LIN {X 0,Y 446.376,Z 609.791,A -85,B 0,C 180,E1 -8740.662,E2 -8740.662} C_VEL
LIN {X 0,Y 447.077,Z 600.807,A -85,B 0,C 180,E1 -8742.253,E2 -8742.253} C_VEL
LIN {X 0,Y 447.648,Z 591.374,A -85,B 0,C 180,E1 -8743.622,E2 -8743.622} C_VEL
LIN {X 0,Y 448.423,Z 580.93,A -85,B 0,C 180,E1 -8744.872,E2 -8744.872} C_VEL
LIN {X 0,Y 449.198,Z 569.398,A -85,B 0,C 180,E1 -8746.008,E2 -8746.008} C_VEL
LIN {X 0,Y 450.087,Z 556.6,A -85,B 0,C 180,E1 -8747.025,E2 -8747.025} C_VEL
LIN {X 0,Y 450.817,Z 543.884,A -85,B 0,C 180,E1 -8747.829,E2 -8747.829} C_VEL
LIN {X 0,Y 451.423,Z 530.193,A -85,B 0,C 180,E1 -8748.495,E2 -8748.495} C_VEL
LIN {X 0,Y 451.967,Z 516.457,A -85,B 0,C 180,E1 -8748.972,E2 -8748.972} C_VEL
LIN {X 0,Y 452.276,Z 502.45,A -85,B 0,C 180,E1 -8749.282,E2 -8749.282} C_VEL
LIN {X 0,Y 453.556,Z 395.078,A -85,B 0,C 180,E1 -8750.999,E2 -8750.999} C_VEL
LIN {X 0,Y 449.146,Z 372.552,A -85,B 0,C 180,E1 -8751.608,E2 -8751.608} C_VEL
LIN {X 0,Y 449.209,Z 369.686,A -85,B 0,C 180,E1 -8752.055,E2 -8752.055} C_VEL
LIN {X 0,Y 449.824,Z 360.532,A -85,B 0,C 180,E1 -8753.724,E2 -8753.724} C_VEL
LIN {X 0,Y 448.206,Z 351.377,A -85,B 0,C 180,E1 -8755.545,E2 -8755.545} C_VEL
LIN {X 0,Y 446.531,Z 343.677,A -85,B 0,C 180,E1 -8757.158,E2 -8757.158} C_VEL
LIN {X 0,Y 446.432,Z 343.497,A -85,B 0,C 180,E1 -8760.25,E2 -8760.25} C_VEL
LIN {X 0,Y 446.449,Z 343.497,A -85,B 0,C 180,E1 -8763.454,E2 -8763.454} C_VEL
LIN {X 0,Y 446.414,Z 343.503,A -85,B 0,C 180,E1 -8766.745,E2 -8766.745} C_VEL
LIN {X 0,Y 446.46,Z 343.497,A -85,B 0,C 180,E1 -8769.526,E2 -8769.526} C_VEL
LIN {X 0,Y 446.433,Z 343.498,A -85,B 0,C 180,E1 -8772.605,E2 -8772.605} C_VEL
LIN {X 0,Y 446.456,Z 343.496,A -85,B 0,C 180,E1 -8775.104,E2 -8775.104} C_VEL
LIN {X 0,Y 446.433,Z 343.501,A -85,B 0,C 180,E1 -8778.609,E2 -8778.609} C_VEL
LIN {X 0,Y 446.448,Z 343.498,A -85,B 0,C 180,E1 -8780.973,E2 -8780.973} C_VEL
LIN {X 0,Y 446.424,Z 343.502,A -85,B 0,C 180,E1 -8784.374,E2 -8784.374} C_VEL
LIN {X 0,Y 446.427,Z 343.504,A -85,B 0,C 180,E1 -8787.639,E2 -8787.639} C_VEL
LIN {X 0,Y 446.477,Z 343.679,A -85,B 0,C 180,E1 -8790.51,E2 -8790.51} C_VEL
LIN {X 0,Y 449.215,Z 353.817,A -85,B 0,C 180,E1 -8792.262,E2 -8792.262} C_VEL
LIN {X 0,Y 450.789,Z 362.335,A -85,B 0,C 180,E1 -8793.62,E2 -8793.62} C_VEL
LIN {X 0,Y 449.985,Z 382.554,A -85,B 0,C 180,E1 -8796.53,E2 -8796.53} C_VEL
LIN {X 0,Y 449.131,Z 404.177,A -85,B 0,C 180,E1 -8799.625,E2 -8799.625} C_VEL
LIN {X 0,Y 448.594,Z 420.532,A -85,B 0,C 180,E1 -8801.952,E2 -8801.952} C_VEL
LIN {X 0,Y 450.781,Z 434.978,A -85,B 0,C 180,E1 -8802.407,E2 -8802.407} C_VEL
LIN {X 0,Y 451.257,Z 439.705,A -85,B 0,C 180,E1 -8802.531,E2 -8802.531} C_VEL
LIN {X 0,Y 449.92,Z 512.596,A -85,B 0,C 180,E1 -8803.961,E2 -8803.961} C_VEL
LIN {X 0,Y 449.624,Z 533.195,A -85,B 0,C 180,E1 -8804.387,E2 -8804.387} C_VEL
LIN {X 0,Y 449.251,Z 545.627,A -85,B 0,C 180,E1 -8804.809,E2 -8804.809} C_VEL
LIN {X 0,Y 448.731,Z 558.542,A -85,B 0,C 180,E1 -8805.43,E2 -8805.43} C_VEL
LIN {X 0,Y 448.238,Z 570.096,A -85,B 0,C 180,E1 -8806.166,E2 -8806.166} C_VEL
LIN {X 0,Y 447.634,Z 582.325,A -85,B 0,C 180,E1 -8807.169,E2 -8807.169} C_VEL
LIN {X 0,Y 447.092,Z 592.458,A -85,B 0,C 180,E1 -8808.209,E2 -8808.209} C_VEL
LIN {X 0,Y 446.575,Z 601.457,A -85,B 0,C 180,E1 -8809.344,E2 -8809.344} C_VEL
LIN {X 0,Y 446.152,Z 610.26,A -85,B 0,C 180,E1 -8810.708,E2 -8810.708} C_VEL
LIN {X 0,Y 445.834,Z 617.287,A -85,B 0,C 180,E1 -8812.072,E2 -8812.072} C_VEL
LIN {X 0,Y 445.581,Z 623.697,A -85,B 0,C 180,E1 -8813.661,E2 -8813.661} C_VEL
LIN {X 0,Y 445.499,Z 627.876,A -85,B 0,C 180,E1 -8815.023,E2 -8815.023} C_VEL
LIN {X 0,Y 445.388,Z 630.958,A -85,B 0,C 180,E1 -8816.381,E2 -8816.381} C_VEL
LIN {X 0,Y 445.405,Z 632.448,A -85,B 0,C 180,E1 -8817.287,E2 -8817.287} C_VEL
LIN {X 0,Y 445.353,Z 633.484,A -85,B 0,C 180,E1 -8818.191,E2 -8818.191} C_VEL
LIN {X 0,Y 445.316,Z 634.118,A -85,B 0,C 180,E1 -8819.096,E2 -8819.096} C_VEL
LIN {X 0,Y 445.293,Z 634.338,A -85,B 0,C 180,E1 -8820,E2 -8820} C_VEL
LIN {X 0,Y 445.316,Z 634.095,A -85,B 0,C 180,E1 -8820.904,E2 -8820.904} C_VEL
LIN {X 0,Y 445.353,Z 633.448,A -85,B 0,C 180,E1 -8821.809,E2 -8821.809} C_VEL
LIN {X 0,Y 445.405,Z 632.398,A -85,B 0,C 180,E1 -8822.713,E2 -8822.713} C_VEL
LIN {X 0,Y 445.384,Z 630.876,A -85,B 0,C 180,E1 -8823.619,E2 -8823.619} C_VEL
LIN {X 0,Y 445.493,Z 627.764,A -85,B 0,C 180,E1 -8824.978,E2 -8824.978} C_VEL
LIN {X 0,Y 445.588,Z 623.157,A -85,B 0,C 180,E1 -8826.449,E2 -8826.449} C_VEL
LIN {X 0,Y 445.797,Z 617.104,A -85,B 0,C 180,E1 -8827.929,E2 -8827.929} C_VEL
LIN {X 0,Y 446.098,Z 610.002,A -85,B 0,C 180,E1 -8829.293,E2 -8829.293} C_VEL
LIN {X 0,Y 446.496,Z 601.134,A -85,B 0,C 180,E1 -8830.658,E2 -8830.658} C_VEL
LIN {X 0,Y 446.983,Z 592.036,A -85,B 0,C 180,E1 -8831.795,E2 -8831.795} C_VEL
LIN {X 0,Y 447.491,Z 581.892,A -85,B 0,C 180,E1 -8832.823,E2 -8832.823} C_VEL
LIN {X 0,Y 447.987,Z 570.879,A -85,B 0,C 180,E1 -8833.726,E2 -8833.726} C_VEL
LIN {X 0,Y 448.466,Z 559.527,A -85,B 0,C 180,E1 -8834.463,E2 -8834.463} C_VEL
LIN {X 0,Y 448.936,Z 546.761,A -85,B 0,C 180,E1 -8835.086,E2 -8835.086} C_VEL
LIN {X 0,Y 449.3,Z 534.57,A -85,B 0,C 180,E1 -8835.509,E2 -8835.509} C_VEL
LIN {X 0,Y 449.505,Z 518.418,A -85,B 0,C 180,E1 -8835.85,E2 -8835.85} C_VEL
LIN {X 0,Y 450.479,Z 437.6,A -85,B 0,C 180,E1 -8837.331,E2 -8837.331} C_VEL
LIN {X 0,Y 448.072,Z 420.918,A -85,B 0,C 180,E1 -8837.745,E2 -8837.745} C_VEL
LIN {X 0,Y 448.866,Z 399.314,A -85,B 0,C 180,E1 -8840.867,E2 -8840.867} C_VEL
LIN {X 0,Y 449.722,Z 378.014,A -85,B 0,C 180,E1 -8843.974,E2 -8843.974} C_VEL
LIN {X 0,Y 450.347,Z 363.098,A -85,B 0,C 180,E1 -8846.159,E2 -8846.159} C_VEL
LIN {X 0,Y 449.696,Z 358.003,A -85,B 0,C 180,E1 -8846.951,E2 -8846.951} C_VEL
LIN {X 0,Y 446.503,Z 343.612,A -85,B 0,C 180,E1 -8849.316,E2 -8849.316} C_VEL
LIN {X 0,Y 446.428,Z 343.504,A -85,B 0,C 180,E1 -8852.361,E2 -8852.361} C_VEL
LIN {X 0,Y 446.425,Z 343.5,A -85,B 0,C 180,E1 -8855.626,E2 -8855.626} C_VEL
LIN {X 0,Y 446.443,Z 343.497,A -85,B 0,C 180,E1 -8859.027,E2 -8859.027} C_VEL
LIN {X 0,Y 446.439,Z 343.5,A -85,B 0,C 180,E1 -8862.277,E2 -8862.277} C_VEL
LIN {X 0,Y 446.456,Z 343.481,A -85,B 0,C 180,E1 -8865.103,E2 -8865.103} C_VEL
LIN {X 0,Y 446.434,Z 343.497,A -85,B 0,C 180,E1 -8868.609,E2 -8868.609} C_VEL
LIN {X 0,Y 446.462,Z 343.491,A -85,B 0,C 180,E1 -8870.974,E2 -8870.974} C_VEL
LIN {X 0,Y 446.426,Z 343.495,A -85,B 0,C 180,E1 -8874.374,E2 -8874.374} C_VEL
LIN {X 0,Y 446.428,Z 343.496,A -85,B 0,C 180,E1 -8877.638,E2 -8877.638} C_VEL
LIN {X 0,Y 446.454,Z 343.474,A -85,B 0,C 180,E1 -8880.79,E2 -8880.79} C_VEL
LIN {X 0,Y 446.534,Z 343.577,A -85,B 0,C 180,E1 -8882.842,E2 -8882.842} C_VEL
LIN {X 0,Y 448.194,Z 351.14,A -85,B 0,C 180,E1 -8884.454,E2 -8884.454} C_VEL
LIN {X 0,Y 449.464,Z 357.575,A -85,B 0,C 180,E1 -8885.747,E2 -8885.747} C_VEL
LIN {X 0,Y 449.036,Z 359.859,A -85,B 0,C 180,E1 -8886.151,E2 -8886.151} C_VEL
LIN {X 0,Y 446.239,Z 363.844,A -85,B 0,C 180,E1 -8886.742,E2 -8886.742} C_VEL
LIN {X 0,Y 443.163,Z 367.892,A -85,B 0,C 180,E1 -8887.336,E2 -8887.336} C_VEL
LIN {X 0,Y 442.357,Z 370.288,A -85,B 0,C 180,E1 -8887.743,E2 -8887.743} C_VEL
LIN {X 0,Y 442.345,Z 372.633,A -85,B 0,C 180,E1 -8888.092,E2 -8888.092} C_VEL
LIN {X 0,Y 446.762,Z 395.118,A -85,B 0,C 180,E1 -8888.712,E2 -8888.712} C_VEL
LIN {X 0,Y 445.847,Z 481.863,A -85,B 0,C 180,E1 -8890.129,E2 -8890.129} C_VEL
LIN {X 0,Y 445.43,Z 510.338,A -85,B 0,C 180,E1 -8890.619,E2 -8890.619} C_VEL
LIN {X 0,Y 444.898,Z 524.682,A -85,B 0,C 180,E1 -8891.044,E2 -8891.044} C_VEL
LIN {X 0,Y 444.37,Z 537.804,A -85,B 0,C 180,E1 -8891.612,E2 -8891.612} C_VEL
LIN {X 0,Y 443.61,Z 551.386,A -85,B 0,C 180,E1 -8892.393,E2 -8892.393} C_VEL
LIN {X 0,Y 442.855,Z 563.522,A -85,B 0,C 180,E1 -8893.282,E2 -8893.282} C_VEL
LIN {X 0,Y 441.938,Z 575.005,A -85,B 0,C 180,E1 -8894.314,E2 -8894.314} C_VEL
LIN {X 0,Y 441.147,Z 585.541,A -85,B 0,C 180,E1 -8895.467,E2 -8895.467} C_VEL
LIN {X 0,Y 440.361,Z 595.567,A -85,B 0,C 180,E1 -8896.791,E2 -8896.791} C_VEL
LIN {X 0,Y 439.776,Z 604.634,A -85,B 0,C 180,E1 -8898.242,E2 -8898.242} C_VEL
LIN {X 0,Y 439.211,Z 612.909,A -85,B 0,C 180,E1 -8899.861,E2 -8899.861} C_VEL
LIN {X 0,Y 438.818,Z 618.678,A -85,B 0,C 180,E1 -8901.247,E2 -8901.247} C_VEL
LIN {X 0,Y 438.526,Z 623.423,A -85,B 0,C 180,E1 -8902.633,E2 -8902.633} C_VEL
LIN {X 0,Y 438.428,Z 628.334,A -85,B 0,C 180,E1 -8904.48,E2 -8904.48} C_VEL
LIN {X 0,Y 438.275,Z 631.757,A -85,B 0,C 180,E1 -8906.321,E2 -8906.321} C_VEL
LIN {X 0,Y 438.273,Z 633.794,A -85,B 0,C 180,E1 -8908.161,E2 -8908.161} C_VEL
LIN {X 0,Y 438.205,Z 634.497,A -85,B 0,C 180,E1 -8909.999,E2 -8909.999} C_VEL
LIN {X 0,Y 438.272,Z 633.874,A -85,B 0,C 180,E1 -8911.837,E2 -8911.837} C_VEL
LIN {X 0,Y 438.274,Z 631.91,A -85,B 0,C 180,E1 -8913.676,E2 -8913.676} C_VEL
LIN {X 0,Y 438.427,Z 628.556,A -85,B 0,C 180,E1 -8915.518,E2 -8915.518} C_VEL
LIN {X 0,Y 438.521,Z 623.713,A -85,B 0,C 180,E1 -8917.365,E2 -8917.365} C_VEL
LIN {X 0,Y 438.93,Z 617.239,A -85,B 0,C 180,E1 -8919.212,E2 -8919.212} C_VEL
LIN {X 0,Y 439.321,Z 610.031,A -85,B 0,C 180,E1 -8920.833,E2 -8920.833} C_VEL
LIN {X 0,Y 440.069,Z 601.116,A -85,B 0,C 180,E1 -8922.449,E2 -8922.449} C_VEL
LIN {X 0,Y 440.7,Z 591.754,A -85,B 0,C 180,E1 -8923.839,E2 -8923.839} C_VEL
LIN {X 0,Y 441.494,Z 581.385,A -85,B 0,C 180,E1 -8925.108,E2 -8925.108} C_VEL
LIN {X 0,Y 442.384,Z 569.949,A -85,B 0,C 180,E1 -8926.259,E2 -8926.259} C_VEL
LIN {X 0,Y 443.21,Z 557.277,A -85,B 0,C 180,E1 -8927.295,E2 -8927.295} C_VEL
LIN {X 0,Y 444.099,Z 543.738,A -85,B 0,C 180,E1 -8928.165,E2 -8928.165} C_VEL
LIN {X 0,Y 444.738,Z 529.988,A -85,B 0,C 180,E1 -8928.841,E2 -8928.841} C_VEL
LIN {X 0,Y 445.286,Z 516.176,A -85,B 0,C 180,E1 -8929.325,E2 -8929.325} C_VEL
LIN {X 0,Y 445.619,Z 501.92,A -85,B 0,C 180,E1 -8929.64,E2 -8929.64} C_VEL
LIN {X 0,Y 446.91,Z 395.787,A -85,B 0,C 180,E1 -8931.364,E2 -8931.364} C_VEL
LIN {X 0,Y 442.305,Z 372.235,A -85,B 0,C 180,E1 -8932.03,E2 -8932.03} C_VEL
LIN {X 0,Y 442.902,Z 360.808,A -85,B 0,C 180,E1 -8934.116,E2 -8934.116} C_VEL
LIN {X 0,Y 440.37,Z 348.452,A -85,B 0,C 180,E1 -8936.655,E2 -8936.655} C_VEL
LIN {X 0,Y 439.506,Z 344.455,A -85,B 0,C 180,E1 -8937.555,E2 -8937.555} C_VEL
LIN {X 0,Y 439.368,Z 344.377,A -85,B 0,C 180,E1 -8940.786,E2 -8940.786} C_VEL
LIN {X 0,Y 439.384,Z 344.38,A -85,B 0,C 180,E1 -8944.042,E2 -8944.042} C_VEL
LIN {X 0,Y 439.36,Z 344.38,A -85,B 0,C 180,E1 -8947.432,E2 -8947.432} C_VEL
LIN {X 0,Y 439.423,Z 344.364,A -85,B 0,C 180,E1 -8949.852,E2 -8949.852} C_VEL
LIN {X 0,Y 439.397,Z 344.375,A -85,B 0,C 180,E1 -8952.629,E2 -8952.629} C_VEL
LIN {X 0,Y 439.397,Z 344.364,A -85,B 0,C 180,E1 -8956.032,E2 -8956.032} C_VEL
LIN {X 0,Y 439.393,Z 344.375,A -85,B 0,C 180,E1 -8959.021,E2 -8959.021} C_VEL
LIN {X 0,Y 439.385,Z 344.358,A -85,B 0,C 180,E1 -8961.604,E2 -8961.604} C_VEL
LIN {X 0,Y 439.393,Z 344.371,A -85,B 0,C 180,E1 -8964.843,E2 -8964.843} C_VEL
LIN {X 0,Y 439.366,Z 344.372,A -85,B 0,C 180,E1 -8968.139,E2 -8968.139} C_VEL
LIN {X 0,Y 439.416,Z 344.343,A -85,B 0,C 180,E1 -8971.326,E2 -8971.326} C_VEL
LIN {X 0,Y 439.403,Z 344.37,A -85,B 0,C 180,E1 -8974.415,E2 -8974.415} C_VEL
LIN {X 0,Y 439.357,Z 344.379,A -85,B 0,C 180,E1 -8977.424,E2 -8977.424} C_VEL
LIN {X 0,Y 439.431,Z 344.368,A -85,B 0,C 180,E1 -8980.662,E2 -8980.662} C_VEL
LIN {X 0,Y 439.452,Z 344.356,A -85,B 0,C 180,E1 -8984.224,E2 -8984.224} C_VEL
LIN {X 0,Y 439.498,Z 344.359,A -85,B 0,C 180,E1 -8988.002,E2 -8988.002} C_VEL
LIN {X 0,Y 439.537,Z 344.354,A -85,B 0,C 180,E1 -8991.726,E2 -8991.726} C_VEL
LIN {X 0,Y 439.614,Z 344.346,A -85,B 0,C 180,E1 -8994.496,E2 -8994.496} C_VEL
LIN {X 0,Y 439.626,Z 344.34,A -85,B 0,C 180,E1 -8998.168,E2 -8998.168} C_VEL
LIN {X 0,Y 439.755,Z 344.329,A -85,B 0,C 180,E1 -9000,E2 -9000} C_VEL
LIN {X 0,Y 439.648,Z 344.338,A -85,B 0,C 180,E1 -9002.749,E2 -9002.749} C_VEL
LIN {X 0,Y 439.61,Z 344.348,A -85,B 0,C 180,E1 -9006.425,E2 -9006.425} C_VEL
LIN {X 0,Y 439.492,Z 344.353,A -85,B 0,C 180,E1 -9009.202,E2 -9009.202} C_VEL
LIN {X 0,Y 439.493,Z 344.366,A -85,B 0,C 180,E1 -9012.727,E2 -9012.727} C_VEL
LIN {X 0,Y 439.436,Z 344.36,A -85,B 0,C 180,E1 -9016.349,E2 -9016.349} C_VEL
LIN {X 0,Y 439.393,Z 344.371,A -85,B 0,C 180,E1 -9019.627,E2 -9019.627} C_VEL
LIN {X 0,Y 439.357,Z 344.378,A -85,B 0,C 180,E1 -9022.576,E2 -9022.576} C_VEL
LIN {X 0,Y 439.403,Z 344.369,A -85,B 0,C 180,E1 -9025.585,E2 -9025.585} C_VEL
LIN {X 0,Y 439.407,Z 344.344,A -85,B 0,C 180,E1 -9028.674,E2 -9028.674} C_VEL
LIN {X 0,Y 439.361,Z 344.374,A -85,B 0,C 180,E1 -9032.031,E2 -9032.031} C_VEL
LIN {X 0,Y 439.387,Z 344.371,A -85,B 0,C 180,E1 -9035.342,E2 -9035.342} C_VEL
LIN {X 0,Y 439.389,Z 344.359,A -85,B 0,C 180,E1 -9038.594,E2 -9038.594} C_VEL
LIN {X 0,Y 439.397,Z 344.374,A -85,B 0,C 180,E1 -9041.26,E2 -9041.26} C_VEL
LIN {X 0,Y 439.403,Z 344.358,A -85,B 0,C 180,E1 -9044.729,E2 -9044.729} C_VEL
LIN {X 0,Y 439.406,Z 344.377,A -85,B 0,C 180,E1 -9047.799,E2 -9047.799} C_VEL
LIN {X 0,Y 439.446,Z 344.361,A -85,B 0,C 180,E1 -9050.231,E2 -9050.231} C_VEL
LIN {X 0,Y 439.372,Z 344.375,A -85,B 0,C 180,E1 -9053.714,E2 -9053.714} C_VEL
LIN {X 0,Y 439.371,Z 344.374,A -85,B 0,C 180,E1 -9057.056,E2 -9057.056} C_VEL
LIN {X 0,Y 439.392,Z 344.356,A -85,B 0,C 180,E1 -9060.277,E2 -9060.277} C_VEL
LIN {X 0,Y 439.514,Z 344.507,A -85,B 0,C 180,E1 -9062.516,E2 -9062.516} C_VEL
LIN {X 0,Y 442.183,Z 357.077,A -85,B 0,C 180,E1 -9065.174,E2 -9065.174} C_VEL
LIN {X 0,Y 442.975,Z 361.879,A -85,B 0,C 180,E1 -9066.137,E2 -9066.137} C_VEL
LIN {X 0,Y 442.309,Z 372.234,A -85,B 0,C 180,E1 -9068.015,E2 -9068.015} C_VEL
LIN {X 0,Y 446.811,Z 395.263,A -85,B 0,C 180,E1 -9068.667,E2 -9068.667} C_VEL
LIN {X 0,Y 445.667,Z 499.235,A -85,B 0,C 180,E1 -9070.363,E2 -9070.363} C_VEL
LIN {X 0,Y 445.33,Z 514.564,A -85,B 0,C 180,E1 -9070.677,E2 -9070.677} C_VEL
LIN {X 0,Y 444.741,Z 528.993,A -85,B 0,C 180,E1 -9071.159,E2 -9071.159} C_VEL
LIN {X 0,Y 444.135,Z 542.56,A -85,B 0,C 180,E1 -9071.811,E2 -9071.811} C_VEL
LIN {X 0,Y 443.37,Z 555.097,A -85,B 0,C 180,E1 -9072.592,E2 -9072.592} C_VEL
LIN {X 0,Y 442.576,Z 566.878,A -85,B 0,C 180,E1 -9073.511,E2 -9073.511} C_VEL
LIN {X 0,Y 441.67,Z 578.84,A -85,B 0,C 180,E1 -9074.662,E2 -9074.662} C_VEL
LIN {X 0,Y 440.831,Z 589.633,A -85,B 0,C 180,E1 -9075.93,E2 -9075.93} C_VEL
LIN {X 0,Y 440.138,Z 599.354,A -85,B 0,C 180,E1 -9077.318,E2 -9077.318} C_VEL
LIN {X 0,Y 439.576,Z 607.419,A -85,B 0,C 180,E1 -9078.707,E2 -9078.707} C_VEL
LIN {X 0,Y 439.034,Z 615.145,A -85,B 0,C 180,E1 -9080.325,E2 -9080.325} C_VEL
LIN {X 0,Y 438.709,Z 620.535,A -85,B 0,C 180,E1 -9081.712,E2 -9081.712} C_VEL
LIN {X 0,Y 438.504,Z 626.208,A -85,B 0,C 180,E1 -9083.56,E2 -9083.56} C_VEL
LIN {X 0,Y 438.33,Z 630.324,A -85,B 0,C 180,E1 -9085.403,E2 -9085.403} C_VEL
LIN {X 0,Y 438.296,Z 633.008,A -85,B 0,C 180,E1 -9087.244,E2 -9087.244} C_VEL
LIN {X 0,Y 438.228,Z 634.335,A -85,B 0,C 180,E1 -9089.082,E2 -9089.082} C_VEL
LIN {X 0,Y 438.228,Z 634.333,A -85,B 0,C 180,E1 -9090.92,E2 -9090.92} C_VEL
LIN {X 0,Y 438.296,Z 632.999,A -85,B 0,C 180,E1 -9092.758,E2 -9092.758} C_VEL
LIN {X 0,Y 438.33,Z 630.311,A -85,B 0,C 180,E1 -9094.599,E2 -9094.599} C_VEL
LIN {X 0,Y 438.465,Z 626.194,A -85,B 0,C 180,E1 -9096.443,E2 -9096.443} C_VEL
LIN {X 0,Y 438.711,Z 620.519,A -85,B 0,C 180,E1 -9098.291,E2 -9098.291} C_VEL
LIN {X 0,Y 439.118,Z 614.115,A -85,B 0,C 180,E1 -9099.908,E2 -9099.908} C_VEL
LIN {X 0,Y 439.69,Z 606.16,A -85,B 0,C 180,E1 -9101.526,E2 -9101.526} C_VEL
LIN {X 0,Y 440.286,Z 596.856,A -85,B 0,C 180,E1 -9103.068,E2 -9103.068} C_VEL
LIN {X 0,Y 440.959,Z 587.809,A -85,B 0,C 180,E1 -9104.303,E2 -9104.303} C_VEL
LIN {X 0,Y 441.827,Z 576.624,A -85,B 0,C 180,E1 -9105.572,E2 -9105.572} C_VEL
LIN {X 0,Y 442.68,Z 565.487,A -85,B 0,C 180,E1 -9106.606,E2 -9106.606} C_VEL
LIN {X 0,Y 443.502,Z 553.358,A -85,B 0,C 180,E1 -9107.524,E2 -9107.524} C_VEL
LIN {X 0,Y 444.242,Z 540.457,A -85,B 0,C 180,E1 -9108.298,E2 -9108.298} C_VEL
LIN {X 0,Y 444.831,Z 526.59,A -85,B 0,C 180,E1 -9108.929,E2 -9108.929} C_VEL
LIN {X 0,Y 445.422,Z 512.051,A -85,B 0,C 180,E1 -9109.381,E2 -9109.381} C_VEL
LIN {X 0,Y 445.768,Z 491.702,A -85,B 0,C 180,E1 -9109.755,E2 -9109.755} C_VEL
LIN {X 0,Y 446.797,Z 395.301,A -85,B 0,C 180,E1 -9111.328,E2 -9111.328} C_VEL
LIN {X 0,Y 442.295,Z 372.483,A -85,B 0,C 180,E1 -9111.964,E2 -9111.964} C_VEL
LIN {X 0,Y 442.39,Z 369.685,A -85,B 0,C 180,E1 -9112.414,E2 -9112.414} C_VEL
LIN {X 0,Y 442.925,Z 361.838,A -85,B 0,C 180,E1 -9113.868,E2 -9113.868} C_VEL
LIN {X 0,Y 441.259,Z 352.683,A -85,B 0,C 180,E1 -9115.724,E2 -9115.724} C_VEL
LIN {X 0,Y 439.48,Z 344.461,A -85,B 0,C 180,E1 -9117.501,E2 -9117.501} C_VEL
LIN {X 0,Y 439.366,Z 344.382,A -85,B 0,C 180,E1 -9120.789,E2 -9120.789} C_VEL
LIN {X 0,Y 439.392,Z 344.379,A -85,B 0,C 180,E1 -9124.044,E2 -9124.044} C_VEL
LIN {X 0,Y 439.362,Z 344.381,A -85,B 0,C 180,E1 -9126.889,E2 -9126.889} C_VEL
LIN {X 0,Y 439.406,Z 344.376,A -85,B 0,C 180,E1 -9129.85,E2 -9129.85} C_VEL
LIN {X 0,Y 439.385,Z 344.376,A -85,B 0,C 180,E1 -9132.627,E2 -9132.627} C_VEL
LIN {X 0,Y 439.404,Z 344.375,A -85,B 0,C 180,E1 -9135.271,E2 -9135.271} C_VEL
LIN {X 0,Y 439.393,Z 344.378,A -85,B 0,C 180,E1 -9138.744,E2 -9138.744} C_VEL
LIN {X 0,Y 439.379,Z 344.381,A -85,B 0,C 180,E1 -9141.608,E2 -9141.608} C_VEL
LIN {X 0,Y 439.404,Z 344.376,A -85,B 0,C 180,E1 -9144.844,E2 -9144.844} C_VEL
LIN {X 0,Y 439.378,Z 344.382,A -85,B 0,C 180,E1 -9148.14,E2 -9148.14} C_VEL
LIN {X 0,Y 439.423,Z 344.584,A -85,B 0,C 180,E1 -9150.047,E2 -9150.047} C_VEL
LIN {X 0,Y 442.588,Z 355.998,A -85,B 0,C 180,E1 -9152.067,E2 -9152.067} C_VEL
LIN {X 0,Y 444.123,Z 364.501,A -85,B 0,C 180,E1 -9153.459,E2 -9153.459} C_VEL
LIN {X 0,Y 443.117,Z 388.214,A -85,B 0,C 180,E1 -9156.913,E2 -9156.913} C_VEL
LIN {X 0,Y 442.013,Z 414.507,A -85,B 0,C 180,E1 -9160.736,E2 -9160.736} C_VEL
LIN {X 0,Y 441.811,Z 420.633,A -85,B 0,C 180,E1 -9161.599,E2 -9161.599} C_VEL
LIN {X 0,Y 444.313,Z 436.885,A -85,B 0,C 180,E1 -9162.118,E2 -9162.118} C_VEL
LIN {X 0,Y 444.594,Z 441.835,A -85,B 0,C 180,E1 -9162.242,E2 -9162.242} C_VEL
LIN {X 0,Y 443.169,Z 512.806,A -85,B 0,C 180,E1 -9163.681,E2 -9163.681} C_VEL
LIN {X 0,Y 442.841,Z 534.049,A -85,B 0,C 180,E1 -9164.141,E2 -9164.141} C_VEL
LIN {X 0,Y 442.384,Z 547.476,A -85,B 0,C 180,E1 -9164.627,E2 -9164.627} C_VEL
LIN {X 0,Y 441.875,Z 559.905,A -85,B 0,C 180,E1 -9165.257,E2 -9165.257} C_VEL
LIN {X 0,Y 441.297,Z 571.839,A -85,B 0,C 180,E1 -9166.062,E2 -9166.062} C_VEL
LIN {X 0,Y 440.724,Z 581.909,A -85,B 0,C 180,E1 -9166.91,E2 -9166.91} C_VEL
LIN {X 0,Y 440.137,Z 592.577,A -85,B 0,C 180,E1 -9168.019,E2 -9168.019} C_VEL
LIN {X 0,Y 439.586,Z 601.564,A -85,B 0,C 180,E1 -9169.172,E2 -9169.172} C_VEL
LIN {X 0,Y 439.123,Z 610.348,A -85,B 0,C 180,E1 -9170.558,E2 -9170.558} C_VEL
LIN {X 0,Y 438.777,Z 617.351,A -85,B 0,C 180,E1 -9171.943,E2 -9171.943} C_VEL
LIN {X 0,Y 438.509,Z 623.756,A -85,B 0,C 180,E1 -9173.559,E2 -9173.559} C_VEL
LIN {X 0,Y 438.434,Z 627.924,A -85,B 0,C 180,E1 -9174.942,E2 -9174.942} C_VEL
LIN {X 0,Y 438.289,Z 630.993,A -85,B 0,C 180,E1 -9176.323,E2 -9176.323} C_VEL
LIN {X 0,Y 438.317,Z 632.467,A -85,B 0,C 180,E1 -9177.243,E2 -9177.243} C_VEL
LIN {X 0,Y 438.275,Z 633.496,A -85,B 0,C 180,E1 -9178.162,E2 -9178.162} C_VEL
LIN {X 0,Y 438.232,Z 634.12,A -85,B 0,C 180,E1 -9179.081,E2 -9179.081} C_VEL
LIN {X 0,Y 438.207,Z 634.321,A -85,B 0,C 180,E1 -9180,E2 -9180} C_VEL
LIN {X 0,Y 438.231,Z 634.063,A -85,B 0,C 180,E1 -9180.919,E2 -9180.919} C_VEL
LIN {X 0,Y 438.275,Z 633.402,A -85,B 0,C 180,E1 -9181.838,E2 -9181.838} C_VEL
LIN {X 0,Y 438.302,Z 632.331,A -85,B 0,C 180,E1 -9182.757,E2 -9182.757} C_VEL
LIN {X 0,Y 438.286,Z 630.781,A -85,B 0,C 180,E1 -9183.678,E2 -9183.678} C_VEL
LIN {X 0,Y 438.406,Z 627.63,A -85,B 0,C 180,E1 -9185.058,E2 -9185.058} C_VEL
LIN {X 0,Y 438.509,Z 623.368,A -85,B 0,C 180,E1 -9186.442,E2 -9186.442} C_VEL
LIN {X 0,Y 438.74,Z 616.862,A -85,B 0,C 180,E1 -9188.057,E2 -9188.057} C_VEL
LIN {X 0,Y 439.064,Z 609.677,A -85,B 0,C 180,E1 -9189.443,E2 -9189.443} C_VEL
LIN {X 0,Y 439.461,Z 600.73,A -85,B 0,C 180,E1 -9190.831,E2 -9190.831} C_VEL
LIN {X 0,Y 440.053,Z 590.462,A -85,B 0,C 180,E1 -9192.1,E2 -9192.1} C_VEL
LIN {X 0,Y 440.627,Z 579.467,A -85,B 0,C 180,E1 -9193.193,E2 -9193.193} C_VEL
LIN {X 0,Y 441.105,Z 568.477,A -85,B 0,C 180,E1 -9194.062,E2 -9194.062} C_VEL
LIN {X 0,Y 441.661,Z 555.324,A -85,B 0,C 180,E1 -9194.868,E2 -9194.868} C_VEL
LIN {X 0,Y 442.162,Z 542.454,A -85,B 0,C 180,E1 -9195.44,E2 -9195.44} C_VEL
LIN {X 0,Y 442.502,Z 529.059,A -85,B 0,C 180,E1 -9195.842,E2 -9195.842} C_VEL
LIN {X 0,Y 443.7,Z 438.826,A -85,B 0,C 180,E1 -9197.539,E2 -9197.539} C_VEL
LIN {X 0,Y 441.144,Z 420.76,A -85,B 0,C 180,E1 -9198.009,E2 -9198.009} C_VEL
LIN {X 0,Y 441.903,Z 400.525,A -85,B 0,C 180,E1 -9200.968,E2 -9200.968} C_VEL
LIN {X 0,Y 442.899,Z 377.435,A -85,B 0,C 180,E1 -9204.367,E2 -9204.367} C_VEL
LIN {X 0,Y 443.459,Z 364.11,A -85,B 0,C 180,E1 -9206.343,E2 -9206.343} C_VEL
LIN {X 0,Y 442.324,Z 357.23,A -85,B 0,C 180,E1 -9207.437,E2 -9207.437} C_VEL
LIN {X 0,Y 439.458,Z 344.498,A -85,B 0,C 180,E1 -9209.557,E2 -9209.557} C_VEL
LIN {X 0,Y 439.378,Z 344.38,A -85,B 0,C 180,E1 -9212.946,E2 -9212.946} C_VEL
LIN {X 0,Y 439.379,Z 344.382,A -85,B 0,C 180,E1 -9216.287,E2 -9216.287} C_VEL
LIN {X 0,Y 439.407,Z 344.375,A -85,B 0,C 180,E1 -9219.849,E2 -9219.849} C_VEL
LIN {X 0,Y 439.386,Z 344.374,A -85,B 0,C 180,E1 -9222.626,E2 -9222.626} C_VEL
LIN {X 0,Y 439.405,Z 344.359,A -85,B 0,C 180,E1 -9225.27,E2 -9225.27} C_VEL
LIN {X 0,Y 439.394,Z 344.373,A -85,B 0,C 180,E1 -9228.743,E2 -9228.743} C_VEL
LIN {X 0,Y 439.39,Z 344.374,A -85,B 0,C 180,E1 -9231.605,E2 -9231.605} C_VEL
LIN {X 0,Y 439.406,Z 344.372,A -85,B 0,C 180,E1 -9234.844,E2 -9234.844} C_VEL
LIN {X 0,Y 439.378,Z 344.378,A -85,B 0,C 180,E1 -9238.139,E2 -9238.139} C_VEL
LIN {X 0,Y 439.438,Z 344.351,A -85,B 0,C 180,E1 -9241.597,E2 -9241.597} C_VEL
LIN {X 0,Y 439.486,Z 344.502,A -85,B 0,C 180,E1 -9242.563,E2 -9242.563} C_VEL
LIN {X 0,Y 442.14,Z 356.89,A -85,B 0,C 180,E1 -9245.186,E2 -9245.186} C_VEL
LIN {X 0,Y 442.91,Z 361.601,A -85,B 0,C 180,E1 -9246.131,E2 -9246.131} C_VEL
LIN {X 0,Y 442.357,Z 370.288,A -85,B 0,C 180,E1 -9247.743,E2 -9247.743} C_VEL
LIN {X 0,Y 443.121,Z 372.145,A -85,B 0,C 180,E1 -9248.027,E2 -9248.027} C_VEL
LIN {X 0,Y 446.207,Z 375.488,A -85,B 0,C 180,E1 -9248.351,E2 -9248.351} C_VEL
LIN {X 0,Y 448.816,Z 379.031,A -85,B 0,C 180,E1 -9248.543,E2 -9248.543} C_VEL
LIN {X 0,Y 449.61,Z 382.103,A -85,B 0,C 180,E1 -9248.635,E2 -9248.635} C_VEL
LIN {X 0,Y 448.993,Z 384.936,A -85,B 0,C 180,E1 -9248.645,E2 -9248.645} C_VEL
LIN {X 0,Y 446.988,Z 388.163,A -85,B 0,C 180,E1 -9248.6,E2 -9248.6} C_VEL
LIN {X 0,Y 442.3,Z 394.273,A -85,B 0,C 180,E1 -9248.472,E2 -9248.472} C_VEL
LIN {X 0,Y 441.279,Z 397.352,A -85,B 0,C 180,E1 -9248.472,E2 -9248.472} C_VEL
LIN {X 0,Y 440.234,Z 401.386,A -85,B 0,C 180,E1 -9248.488,E2 -9248.488} C_VEL
LIN {X 0,Y 438.781,Z 509.193,A -85,B 0,C 180,E1 -9250.283,E2 -9250.283} C_VEL
LIN {X 0,Y 438.219,Z 523.931,A -85,B 0,C 180,E1 -9250.713,E2 -9250.713} C_VEL
LIN {X 0,Y 437.677,Z 536.806,A -85,B 0,C 180,E1 -9251.266,E2 -9251.266} C_VEL
LIN {X 0,Y 436.895,Z 550.297,A -85,B 0,C 180,E1 -9252.038,E2 -9252.038} C_VEL
LIN {X 0,Y 436.041,Z 563.527,A -85,B 0,C 180,E1 -9253.013,E2 -9253.013} C_VEL
LIN {X 0,Y 435.082,Z 575.009,A -85,B 0,C 180,E1 -9254.06,E2 -9254.06} C_VEL
LIN {X 0,Y 434.245,Z 585.544,A -85,B 0,C 180,E1 -9255.231,E2 -9255.231} C_VEL
LIN {X 0,Y 433.372,Z 596.17,A -85,B 0,C 180,E1 -9256.662,E2 -9256.662} C_VEL
LIN {X 0,Y 432.805,Z 604.636,A -85,B 0,C 180,E1 -9258.05,E2 -9258.05} C_VEL
LIN {X 0,Y 432.156,Z 612.911,A -85,B 0,C 180,E1 -9259.694,E2 -9259.694} C_VEL
LIN {X 0,Y 431.786,Z 618.68,A -85,B 0,C 180,E1 -9261.104,E2 -9261.104} C_VEL
LIN {X 0,Y 431.479,Z 623.425,A -85,B 0,C 180,E1 -9262.512,E2 -9262.512} C_VEL
LIN {X 0,Y 431.327,Z 628.335,A -85,B 0,C 180,E1 -9264.388,E2 -9264.388} C_VEL
LIN {X 0,Y 431.182,Z 631.757,A -85,B 0,C 180,E1 -9266.261,E2 -9266.261} C_VEL
LIN {X 0,Y 431.196,Z 633.795,A -85,B 0,C 180,E1 -9268.131,E2 -9268.131} C_VEL
LIN {X 0,Y 431.121,Z 634.497,A -85,B 0,C 180,E1 -9269.999,E2 -9269.999} C_VEL
LIN {X 0,Y 431.195,Z 633.873,A -85,B 0,C 180,E1 -9271.867,E2 -9271.867} C_VEL
LIN {X 0,Y 431.181,Z 631.909,A -85,B 0,C 180,E1 -9273.737,E2 -9273.737} C_VEL
LIN {X 0,Y 431.325,Z 628.555,A -85,B 0,C 180,E1 -9275.609,E2 -9275.609} C_VEL
LIN {X 0,Y 431.474,Z 623.712,A -85,B 0,C 180,E1 -9277.486,E2 -9277.486} C_VEL
LIN {X 0,Y 431.886,Z 617.237,A -85,B 0,C 180,E1 -9279.364,E2 -9279.364} C_VEL
LIN {X 0,Y 432.317,Z 610.029,A -85,B 0,C 180,E1 -9281.011,E2 -9281.011} C_VEL
LIN {X 0,Y 432.989,Z 602.475,A -85,B 0,C 180,E1 -9282.418,E2 -9282.418} C_VEL
LIN {X 0,Y 433.637,Z 593.57,A -85,B 0,C 180,E1 -9283.806,E2 -9283.806} C_VEL
LIN {X 0,Y 434.345,Z 584.377,A -85,B 0,C 180,E1 -9285.003,E2 -9285.003} C_VEL
LIN {X 0,Y 435.204,Z 573.603,A -85,B 0,C 180,E1 -9286.173,E2 -9286.173} C_VEL
LIN {X 0,Y 436.129,Z 561.821,A -85,B 0,C 180,E1 -9287.222,E2 -9287.222} C_VEL
LIN {X 0,Y 436.972,Z 549.604,A -85,B 0,C 180,E1 -9288.101,E2 -9288.101} C_VEL
LIN {X 0,Y 437.697,Z 536.337,A -85,B 0,C 180,E1 -9288.852,E2 -9288.852} C_VEL
LIN {X 0,Y 438.339,Z 522.526,A -85,B 0,C 180,E1 -9289.431,E2 -9289.431} C_VEL
LIN {X 0,Y 438.86,Z 508.026,A -85,B 0,C 180,E1 -9289.833,E2 -9289.833} C_VEL
LIN {X 0,Y 440.267,Z 396.537,A -85,B 0,C 180,E1 -9291.689,E2 -9291.689} C_VEL
LIN {X 0,Y 435.447,Z 372.318,A -85,B 0,C 180,E1 -9292.388,E2 -9292.388} C_VEL
LIN {X 0,Y 436.06,Z 363.421,A -85,B 0,C 180,E1 -9294.012,E2 -9294.012} C_VEL
LIN {X 0,Y 434.406,Z 354.265,A -85,B 0,C 180,E1 -9295.899,E2 -9295.899} C_VEL
LIN {X 0,Y 432.444,Z 345.358,A -85,B 0,C 180,E1 -9297.854,E2 -9297.854} C_VEL
LIN {X 0,Y 432.367,Z 345.242,A -85,B 0,C 180,E1 -9300.514,E2 -9300.514} C_VEL
LIN {X 0,Y 432.356,Z 345.255,A -85,B 0,C 180,E1 -9304.002,E2 -9304.002} C_VEL
LIN {X 0,Y 432.33,Z 345.255,A -85,B 0,C 180,E1 -9307.198,E2 -9307.198} C_VEL
LIN {X 0,Y 432.353,Z 345.244,A -85,B 0,C 180,E1 -9310.182,E2 -9310.182} C_VEL
LIN {X 0,Y 432.359,Z 345.251,A -85,B 0,C 180,E1 -9313.054,E2 -9313.054} C_VEL
LIN {X 0,Y 432.371,Z 345.235,A -85,B 0,C 180,E1 -9315.657,E2 -9315.657} C_VEL
LIN {X 0,Y 432.366,Z 345.251,A -85,B 0,C 180,E1 -9318.391,E2 -9318.391} C_VEL
LIN {X 0,Y 432.345,Z 345.231,A -85,B 0,C 180,E1 -9321.851,E2 -9321.851} C_VEL
LIN {X 0,Y 432.333,Z 345.253,A -85,B 0,C 180,E1 -9325.322,E2 -9325.322} C_VEL
LIN {X 0,Y 432.315,Z 345.248,A -85,B 0,C 180,E1 -9328.653,E2 -9328.653} C_VEL
LIN {X 0,Y 432.372,Z 345.219,A -85,B 0,C 180,E1 -9331.368,E2 -9331.368} C_VEL
LIN {X 0,Y 432.359,Z 345.25,A -85,B 0,C 180,E1 -9333.967,E2 -9333.967} C_VEL
LIN {X 0,Y 432.311,Z 345.259,A -85,B 0,C 180,E1 -9337.035,E2 -9337.035} C_VEL
LIN {X 0,Y 432.377,Z 345.246,A -85,B 0,C 180,E1 -9340.514,E2 -9340.514} C_VEL
LIN {X 0,Y 432.42,Z 345.233,A -85,B 0,C 180,E1 -9343.961,E2 -9343.961} C_VEL
LIN {X 0,Y 432.471,Z 345.236,A -85,B 0,C 180,E1 -9347.804,E2 -9347.804} C_VEL
LIN {X 0,Y 432.481,Z 345.234,A -85,B 0,C 180,E1 -9351.59,E2 -9351.59} C_VEL
LIN {X 0,Y 432.59,Z 345.221,A -85,B 0,C 180,E1 -9354.406,E2 -9354.406} C_VEL
LIN {X 0,Y 432.596,Z 345.216,A -85,B 0,C 180,E1 -9358.138,E2 -9358.138} C_VEL
LIN {X 0,Y 432.726,Z 345.205,A -85,B 0,C 180,E1 -9360,E2 -9360} C_VEL
LIN {X 0,Y 432.597,Z 345.215,A -85,B 0,C 180,E1 -9362.794,E2 -9362.794} C_VEL
LIN {X 0,Y 432.564,Z 345.227,A -85,B 0,C 180,E1 -9366.53,E2 -9366.53} C_VEL
LIN {X 0,Y 432.435,Z 345.23,A -85,B 0,C 180,E1 -9369.353,E2 -9369.353} C_VEL
LIN {X 0,Y 432.434,Z 345.244,A -85,B 0,C 180,E1 -9372.812,E2 -9372.812} C_VEL
LIN {X 0,Y 432.401,Z 345.237,A -85,B 0,C 180,E1 -9376.479,E2 -9376.479} C_VEL
LIN {X 0,Y 432.331,Z 345.251,A -85,B 0,C 180,E1 -9379.961,E2 -9379.961} C_VEL
LIN {X 0,Y 432.311,Z 345.259,A -85,B 0,C 180,E1 -9382.965,E2 -9382.965} C_VEL
LIN {X 0,Y 432.358,Z 345.249,A -85,B 0,C 180,E1 -9386.033,E2 -9386.033} C_VEL
LIN {X 0,Y 432.333,Z 345.223,A -85,B 0,C 180,E1 -9389.188,E2 -9389.188} C_VEL
LIN {X 0,Y 432.314,Z 345.257,A -85,B 0,C 180,E1 -9392.444,E2 -9392.444} C_VEL
LIN {X 0,Y 432.337,Z 345.25,A -85,B 0,C 180,E1 -9395.633,E2 -9395.633} C_VEL
LIN {X 0,Y 432.351,Z 345.236,A -85,B 0,C 180,E1 -9398.719,E2 -9398.719} C_VEL
LIN {X 0,Y 432.366,Z 345.253,A -85,B 0,C 180,E1 -9401.793,E2 -9401.793} C_VEL
LIN {X 0,Y 432.371,Z 345.235,A -85,B 0,C 180,E1 -9404.343,E2 -9404.343} C_VEL
LIN {X 0,Y 432.359,Z 345.251,A -85,B 0,C 180,E1 -9407.01,E2 -9407.01} C_VEL
LIN {X 0,Y 432.352,Z 345.244,A -85,B 0,C 180,E1 -9409.818,E2 -9409.818} C_VEL
LIN {X 0,Y 432.312,Z 345.256,A -85,B 0,C 180,E1 -9413.024,E2 -9413.024} C_VEL
LIN {X 0,Y 432.355,Z 345.256,A -85,B 0,C 180,E1 -9415.998,E2 -9415.998} C_VEL
LIN {X 0,Y 432.391,Z 345.234,A -85,B 0,C 180,E1 -9419.745,E2 -9419.745} C_VEL
LIN {X 0,Y 432.459,Z 345.396,A -85,B 0,C 180,E1 -9422.213,E2 -9422.213} C_VEL
LIN {X 0,Y 435.023,Z 357.318,A -85,B 0,C 180,E1 -9424.784,E2 -9424.784} C_VEL
LIN {X 0,Y 436.077,Z 363.189,A -85,B 0,C 180,E1 -9425.989,E2 -9425.989} C_VEL
LIN {X 0,Y 435.446,Z 372.228,A -85,B 0,C 180,E1 -9427.649,E2 -9427.649} C_VEL
LIN {X 0,Y 439.189,Z 390.904,A -85,B 0,C 180,E1 -9428.203,E2 -9428.203} C_VEL
LIN {X 0,Y 440.306,Z 397.29,A -85,B 0,C 180,E1 -9428.371,E2 -9428.371} C_VEL
LIN {X 0,Y 438.809,Z 508.803,A -85,B 0,C 180,E1 -9430.226,E2 -9430.226} C_VEL
LIN {X 0,Y 438.333,Z 522.936,A -85,B 0,C 180,E1 -9430.63,E2 -9430.63} C_VEL
LIN {X 0,Y 437.787,Z 535.489,A -85,B 0,C 180,E1 -9431.152,E2 -9431.152} C_VEL
LIN {X 0,Y 437.052,Z 548.69,A -85,B 0,C 180,E1 -9431.885,E2 -9431.885} C_VEL
LIN {X 0,Y 436.225,Z 561.29,A -85,B 0,C 180,E1 -9432.782,E2 -9432.782} C_VEL
LIN {X 0,Y 435.267,Z 573.164,A -85,B 0,C 180,E1 -9433.829,E2 -9433.829} C_VEL
LIN {X 0,Y 434.365,Z 584.011,A -85,B 0,C 180,E1 -9434.998,E2 -9434.998} C_VEL
LIN {X 0,Y 433.582,Z 593.264,A -85,B 0,C 180,E1 -9436.193,E2 -9436.193} C_VEL
LIN {X 0,Y 433.036,Z 602.219,A -85,B 0,C 180,E1 -9437.583,E2 -9437.583} C_VEL
LIN {X 0,Y 432.282,Z 610.933,A -85,B 0,C 180,E1 -9439.226,E2 -9439.226} C_VEL
LIN {X 0,Y 431.886,Z 617.065,A -85,B 0,C 180,E1 -9440.636,E2 -9440.636} C_VEL
LIN {X 0,Y 431.473,Z 623.576,A -85,B 0,C 180,E1 -9442.514,E2 -9442.514} C_VEL
LIN {X 0,Y 431.407,Z 626.565,A -85,B 0,C 180,E1 -9443.588,E2 -9443.588} C_VEL
LIN {X 0,Y 431.258,Z 630.325,A -85,B 0,C 180,E1 -9445.327,E2 -9445.327} C_VEL
LIN {X 0,Y 431.193,Z 633.008,A -85,B 0,C 180,E1 -9447.199,E2 -9447.199} C_VEL
LIN {X 0,Y 431.146,Z 634.335,A -85,B 0,C 180,E1 -9449.067,E2 -9449.067} C_VEL
LIN {X 0,Y 431.146,Z 634.333,A -85,B 0,C 180,E1 -9450.935,E2 -9450.935} C_VEL
LIN {X 0,Y 431.193,Z 632.999,A -85,B 0,C 180,E1 -9452.804,E2 -9452.804} C_VEL
LIN {X 0,Y 431.259,Z 630.31,A -85,B 0,C 180,E1 -9454.675,E2 -9454.675} C_VEL
LIN {X 0,Y 431.38,Z 626.193,A -85,B 0,C 180,E1 -9456.55,E2 -9456.55} C_VEL
LIN {X 0,Y 431.653,Z 620.518,A -85,B 0,C 180,E1 -9458.427,E2 -9458.427} C_VEL
LIN {X 0,Y 432.089,Z 614.114,A -85,B 0,C 180,E1 -9460.071,E2 -9460.071} C_VEL
LIN {X 0,Y 432.689,Z 606.158,A -85,B 0,C 180,E1 -9461.715,E2 -9461.715} C_VEL
LIN {X 0,Y 433.259,Z 597.833,A -85,B 0,C 180,E1 -9463.127,E2 -9463.127} C_VEL
LIN {X 0,Y 434.043,Z 587.807,A -85,B 0,C 180,E1 -9464.536,E2 -9464.536} C_VEL
LIN {X 0,Y 434.968,Z 576.621,A -85,B 0,C 180,E1 -9465.824,E2 -9465.824} C_VEL
LIN {X 0,Y 435.974,Z 564.059,A -85,B 0,C 180,E1 -9466.99,E2 -9466.99} C_VEL
LIN {X 0,Y 436.846,Z 551.043,A -85,B 0,C 180,E1 -9467.958,E2 -9467.958} C_VEL
LIN {X 0,Y 437.658,Z 537.643,A -85,B 0,C 180,E1 -9468.734,E2 -9468.734} C_VEL
LIN {X 0,Y 438.258,Z 523.534,A -85,B 0,C 180,E1 -9469.346,E2 -9469.346} C_VEL
LIN {X 0,Y 438.758,Z 509.759,A -85,B 0,C 180,E1 -9469.749,E2 -9469.749} C_VEL
LIN {X 0,Y 440.055,Z 415.331,A -85,B 0,C 180,E1 -9471.327,E2 -9471.327} C_VEL
LIN {X 0,Y 440.204,Z 396.385,A -85,B 0,C 180,E1 -9471.645,E2 -9471.645} C_VEL
LIN {X 0,Y 435.459,Z 372.53,A -85,B 0,C 180,E1 -9472.325,E2 -9472.325} C_VEL
LIN {X 0,Y 435.594,Z 369.683,A -85,B 0,C 180,E1 -9472.783,E2 -9472.783} C_VEL
LIN {X 0,Y 436.024,Z 363.144,A -85,B 0,C 180,E1 -9474.017,E2 -9474.017} C_VEL
LIN {X 0,Y 434.102,Z 352.777,A -85,B 0,C 180,E1 -9476.161,E2 -9476.161} C_VEL
LIN {X 0,Y 432.464,Z 345.383,A -85,B 0,C 180,E1 -9477.789,E2 -9477.789} C_VEL
LIN {X 0,Y 432.326,Z 345.258,A -85,B 0,C 180,E1 -9481.347,E2 -9481.347} C_VEL
LIN {X 0,Y 432.346,Z 345.255,A -85,B 0,C 180,E1 -9484.678,E2 -9484.678} C_VEL
LIN {X 0,Y 432.35,Z 345.256,A -85,B 0,C 180,E1 -9488.15,E2 -9488.15} C_VEL
LIN {X 0,Y 432.337,Z 345.255,A -85,B 0,C 180,E1 -9491.603,E2 -9491.603} C_VEL
LIN {X 0,Y 432.338,Z 345.255,A -85,B 0,C 180,E1 -9494.348,E2 -9494.348} C_VEL
LIN {X 0,Y 432.325,Z 345.258,A -85,B 0,C 180,E1 -9497.016,E2 -9497.016} C_VEL
LIN {X 0,Y 432.338,Z 345.257,A -85,B 0,C 180,E1 -9499.821,E2 -9499.821} C_VEL
LIN {X 0,Y 432.311,Z 345.261,A -85,B 0,C 180,E1 -9503.022,E2 -9503.022} C_VEL
LIN {X 0,Y 432.364,Z 345.255,A -85,B 0,C 180,E1 -9505.997,E2 -9505.997} C_VEL
LIN {X 0,Y 432.371,Z 345.483,A -85,B 0,C 180,E1 -9509.532,E2 -9509.532} C_VEL
LIN {X 0,Y 435.322,Z 355.477,A -85,B 0,C 180,E1 -9511.379,E2 -9511.379} C_VEL
LIN {X 0,Y 437.376,Z 365.334,A -85,B 0,C 180,E1 -9513.061,E2 -9513.061} C_VEL
LIN {X 0,Y 437.195,Z 372.826,A -85,B 0,C 180,E1 -9514.187,E2 -9514.187} C_VEL
LIN {X 0,Y 436.124,Z 395.269,A -85,B 0,C 180,E1 -9517.498,E2 -9517.498} C_VEL
LIN {X 0,Y 435.077,Z 420.535,A -85,B 0,C 180,E1 -9521.199,E2 -9521.199} C_VEL
LIN {X 0,Y 437.376,Z 434.703,A -85,B 0,C 180,E1 -9521.69,E2 -9521.69} C_VEL
LIN {X 0,Y 438.063,Z 441.166,A -85,B 0,C 180,E1 -9521.878,E2 -9521.878} C_VEL
LIN {X 0,Y 436.527,Z 511.99,A -85,B 0,C 180,E1 -9523.365,E2 -9523.365} C_VEL
LIN {X 0,Y 436.089,Z 534.19,A -85,B 0,C 180,E1 -9523.859,E2 -9523.859} C_VEL
LIN {X 0,Y 435.627,Z 546.849,A -85,B 0,C 180,E1 -9524.322,E2 -9524.322} C_VEL
LIN {X 0,Y 435.082,Z 558.369,A -85,B 0,C 180,E1 -9524.902,E2 -9524.902} C_VEL
LIN {X 0,Y 434.472,Z 570.66,A -85,B 0,C 180,E1 -9525.719,E2 -9525.719} C_VEL
LIN {X 0,Y 433.79,Z 582.564,A -85,B 0,C 180,E1 -9526.735,E2 -9526.735} C_VEL
LIN {X 0,Y 433.191,Z 592.771,A -85,B 0,C 180,E1 -9527.824,E2 -9527.824} C_VEL
LIN {X 0,Y 432.607,Z 601.72,A -85,B 0,C 180,E1 -9528.995,E2 -9528.995} C_VEL
LIN {X 0,Y 432.112,Z 610.473,A -85,B 0,C 180,E1 -9530.404,E2 -9530.404} C_VEL
LIN {X 0,Y 431.736,Z 617.448,A -85,B 0,C 180,E1 -9531.811,E2 -9531.811} C_VEL
LIN {X 0,Y 431.443,Z 623.841,A -85,B 0,C 180,E1 -9533.453,E2 -9533.453} C_VEL
LIN {X 0,Y 431.368,Z 627.99,A -85,B 0,C 180,E1 -9534.859,E2 -9534.859} C_VEL
LIN {X 0,Y 431.196,Z 631.04,A -85,B 0,C 180,E1 -9536.262,E2 -9536.262} C_VEL
LIN {X 0,Y 431.214,Z 632.493,A -85,B 0,C 180,E1 -9537.198,E2 -9537.198} C_VEL
LIN {X 0,Y 431.199,Z 633.512,A -85,B 0,C 180,E1 -9538.132,E2 -9538.132} C_VEL
LIN {X 0,Y 431.15,Z 634.126,A -85,B 0,C 180,E1 -9539.066,E2 -9539.066} C_VEL
LIN {X 0,Y 431.123,Z 634.3,A -85,B 0,C 180,E1 -9540,E2 -9540} C_VEL
LIN {X 0,Y 431.15,Z 634.027,A -85,B 0,C 180,E1 -9540.934,E2 -9540.934} C_VEL
LIN {X 0,Y 431.199,Z 633.349,A -85,B 0,C 180,E1 -9541.868,E2 -9541.868} C_VEL
LIN {X 0,Y 431.199,Z 632.249,A -85,B 0,C 180,E1 -9542.803,E2 -9542.803} C_VEL
LIN {X 0,Y 431.224,Z 629.745,A -85,B 0,C 180,E1 -9544.206,E2 -9544.206} C_VEL
LIN {X 0,Y 431.342,Z 626.186,A -85,B 0,C 180,E1 -9545.61,E2 -9545.61} C_VEL
LIN {X 0,Y 431.473,Z 621.466,A -85,B 0,C 180,E1 -9547.017,E2 -9547.017} C_VEL
LIN {X 0,Y 431.782,Z 614.331,A -85,B 0,C 180,E1 -9548.659,E2 -9548.659} C_VEL
LIN {X 0,Y 432.166,Z 606.523,A -85,B 0,C 180,E1 -9550.068,E2 -9550.068} C_VEL
LIN {X 0,Y 432.558,Z 598.526,A -85,B 0,C 180,E1 -9551.243,E2 -9551.243} C_VEL
LIN {X 0,Y 433.118,Z 588.809,A -85,B 0,C 180,E1 -9552.416,E2 -9552.416} C_VEL
LIN {X 0,Y 433.656,Z 577.721,A -85,B 0,C 180,E1 -9553.494,E2 -9553.494} C_VEL
LIN {X 0,Y 434.217,Z 565.818,A -85,B 0,C 180,E1 -9554.41,E2 -9554.41} C_VEL
LIN {X 0,Y 434.759,Z 554.061,A -85,B 0,C 180,E1 -9555.11,E2 -9555.11} C_VEL
LIN {X 0,Y 435.239,Z 539.873,A -85,B 0,C 180,E1 -9555.722,E2 -9555.722} C_VEL
LIN {X 0,Y 435.625,Z 527.603,A -85,B 0,C 180,E1 -9556.069,E2 -9556.069} C_VEL
LIN {X 0,Y 436.771,Z 439.176,A -85,B 0,C 180,E1 -9557.778,E2 -9557.778} C_VEL
LIN {X 0,Y 434.196,Z 420.726,A -85,B 0,C 180,E1 -9558.268,E2 -9558.268} C_VEL
LIN {X 0,Y 435.012,Z 400.05,A -85,B 0,C 180,E1 -9561.316,E2 -9561.316} C_VEL
LIN {X 0,Y 436.071,Z 376.845,A -85,B 0,C 180,E1 -9564.774,E2 -9564.774} C_VEL
LIN {X 0,Y 436.546,Z 365.065,A -85,B 0,C 180,E1 -9566.536,E2 -9566.536} C_VEL
LIN {X 0,Y 434.552,Z 354.707,A -85,B 0,C 180,E1 -9568.214,E2 -9568.214} C_VEL
LIN {X 0,Y 432.379,Z 345.359,A -85,B 0,C 180,E1 -9569.82,E2 -9569.82} C_VEL
LIN {X 0,Y 432.345,Z 345.255,A -85,B 0,C 180,E1 -9573.552,E2 -9573.552} C_VEL
LIN {X 0,Y 432.343,Z 345.255,A -85,B 0,C 180,E1 -9575.817,E2 -9575.817} C_VEL
LIN {X 0,Y 432.332,Z 345.254,A -85,B 0,C 180,E1 -9579.345,E2 -9579.345} C_VEL
LIN {X 0,Y 432.338,Z 345.256,A -85,B 0,C 180,E1 -9581.797,E2 -9581.797} C_VEL
LIN {X 0,Y 432.339,Z 345.24,A -85,B 0,C 180,E1 -9584.347,E2 -9584.347} C_VEL
LIN {X 0,Y 432.325,Z 345.256,A -85,B 0,C 180,E1 -9587.015,E2 -9587.015} C_VEL
LIN {X 0,Y 432.338,Z 345.247,A -85,B 0,C 180,E1 -9589.82,E2 -9589.82} C_VEL
LIN {X 0,Y 432.321,Z 345.256,A -85,B 0,C 180,E1 -9593.022,E2 -9593.022} C_VEL
LIN {X 0,Y 432.365,Z 345.256,A -85,B 0,C 180,E1 -9595.996,E2 -9595.996} C_VEL
LIN {X 0,Y 432.353,Z 345.246,A -85,B 0,C 180,E1 -9599.489,E2 -9599.489} C_VEL
LIN {X 0,Y 432.483,Z 345.422,A -85,B 0,C 180,E1 -9602.278,E2 -9602.278} C_VEL
LIN {X 0,Y 435.377,Z 358.989,A -85,B 0,C 180,E1 -9605.183,E2 -9605.183} C_VEL
LIN {X 0,Y 436.014,Z 364.218,A -85,B 0,C 180,E1 -9606.235,E2 -9606.235} C_VEL
LIN {X 0,Y 435.466,Z 372.131,A -85,B 0,C 180,E1 -9607.69,E2 -9607.69} C_VEL
LIN {X 0,Y 436.658,Z 378.261,A -85,B 0,C 180,E1 -9607.901,E2 -9607.901} C_VEL
LIN {X 0,Y 440.196,Z 396.396,A -85,B 0,C 180,E1 -9608.4,E2 -9608.4} C_VEL
LIN {X 0,Y 440.234,Z 401.386,A -85,B 0,C 180,E1 -9608.488,E2 -9608.488} C_VEL
LIN {X 0,Y 439.521,Z 407.237,A -85,B 0,C 180,E1 -9608.552,E2 -9608.552} C_VEL
LIN {X 0,Y 433.887,Z 426.269,A -85,B 0,C 180,E1 -9608.591,E2 -9608.591} C_VEL
LIN {X 0,Y 433.244,Z 432.116,A -85,B 0,C 180,E1 -9608.659,E2 -9608.659} C_VEL
LIN {X 0,Y 432.118,Z 509.212,A -85,B 0,C 180,E1 -9609.966,E2 -9609.966} C_VEL
LIN {X 0,Y 431.516,Z 523.943,A -85,B 0,C 180,E1 -9610.402,E2 -9610.402} C_VEL
LIN {X 0,Y 430.97,Z 536.815,A -85,B 0,C 180,E1 -9610.964,E2 -9610.964} C_VEL
LIN {X 0,Y 430.139,Z 550.486,A -85,B 0,C 180,E1 -9611.758,E2 -9611.758} C_VEL
LIN {X 0,Y 429.229,Z 563.533,A -85,B 0,C 180,E1 -9612.735,E2 -9612.735} C_VEL
LIN {X 0,Y 428.222,Z 575.014,A -85,B 0,C 180,E1 -9613.798,E2 -9613.798} C_VEL
LIN {X 0,Y 427.375,Z 585.548,A -85,B 0,C 180,E1 -9614.988,E2 -9614.988} C_VEL
LIN {X 0,Y 426.41,Z 596.173,A -85,B 0,C 180,E1 -9616.44,E2 -9616.44} C_VEL
LIN {X 0,Y 425.835,Z 604.639,A -85,B 0,C 180,E1 -9617.852,E2 -9617.852} C_VEL
LIN {X 0,Y 425.109,Z 612.913,A -85,B 0,C 180,E1 -9619.521,E2 -9619.521} C_VEL
LIN {X 0,Y 424.742,Z 618.682,A -85,B 0,C 180,E1 -9620.955,E2 -9620.955} C_VEL
LIN {X 0,Y 424.403,Z 623.426,A -85,B 0,C 180,E1 -9622.386,E2 -9622.386} C_VEL
LIN {X 0,Y 424.236,Z 628.336,A -85,B 0,C 180,E1 -9624.294,E2 -9624.294} C_VEL
LIN {X 0,Y 424.093,Z 631.758,A -85,B 0,C 180,E1 -9626.198,E2 -9626.198} C_VEL
LIN {X 0,Y 424.121,Z 633.795,A -85,B 0,C 180,E1 -9628.1,E2 -9628.1} C_VEL
LIN {X 0,Y 424.041,Z 634.497,A -85,B 0,C 180,E1 -9629.999,E2 -9629.999} C_VEL
LIN {X 0,Y 424.12,Z 633.873,A -85,B 0,C 180,E1 -9631.898,E2 -9631.898} C_VEL
LIN {X 0,Y 424.092,Z 631.909,A -85,B 0,C 180,E1 -9633.8,E2 -9633.8} C_VEL
LIN {X 0,Y 424.232,Z 628.554,A -85,B 0,C 180,E1 -9635.703,E2 -9635.703} C_VEL
LIN {X 0,Y 424.397,Z 623.711,A -85,B 0,C 180,E1 -9637.612,E2 -9637.612} C_VEL
LIN {X 0,Y 424.717,Z 619.043,A -85,B 0,C 180,E1 -9639.043,E2 -9639.043} C_VEL
LIN {X 0,Y 425.151,Z 612.258,A -85,B 0,C 180,E1 -9640.716,E2 -9640.716} C_VEL
LIN {X 0,Y 425.789,Z 605.176,A -85,B 0,C 180,E1 -9642.147,E2 -9642.147} C_VEL
LIN {X 0,Y 426.441,Z 596.809,A -85,B 0,C 180,E1 -9643.557,E2 -9643.557} C_VEL
LIN {X 0,Y 427.305,Z 586.324,A -85,B 0,C 180,E1 -9645.012,E2 -9645.012} C_VEL
LIN {X 0,Y 428.261,Z 574.772,A -85,B 0,C 180,E1 -9646.32,E2 -9646.32} C_VEL
LIN {X 0,Y 429.233,Z 563.24,A -85,B 0,C 180,E1 -9647.385,E2 -9647.385} C_VEL
LIN {X 0,Y 430.145,Z 551.044,A -85,B 0,C 180,E1 -9648.297,E2 -9648.297} C_VEL
LIN {X 0,Y 430.907,Z 537.459,A -85,B 0,C 180,E1 -9649.098,E2 -9649.098} C_VEL
LIN {X 0,Y 431.619,Z 523.289,A -85,B 0,C 180,E1 -9649.715,E2 -9649.715} C_VEL
LIN {X 0,Y 432.149,Z 509.4,A -85,B 0,C 180,E1 -9650.123,E2 -9650.123} C_VEL
LIN {X 0,Y 433.698,Z 398.117,A -85,B 0,C 180,E1 -9652.006,E2 -9652.006} C_VEL
LIN {X 0,Y 428.974,Z 374.071,A -85,B 0,C 180,E1 -9652.688,E2 -9652.688} C_VEL
LIN {X 0,Y 428.612,Z 371.875,A -85,B 0,C 180,E1 -9652.817,E2 -9652.817} C_VEL
LIN {X 0,Y 429.179,Z 364.727,A -85,B 0,C 180,E1 -9654.165,E2 -9654.165} C_VEL
LIN {X 0,Y 426.825,Z 352.518,A -85,B 0,C 180,E1 -9656.746,E2 -9656.746} C_VEL
LIN {X 0,Y 425.374,Z 346.21,A -85,B 0,C 180,E1 -9658.19,E2 -9658.19} C_VEL
LIN {X 0,Y 425.298,Z 346.128,A -85,B 0,C 180,E1 -9660.813,E2 -9660.813} C_VEL
LIN {X 0,Y 425.308,Z 346.134,A -85,B 0,C 180,E1 -9664.287,E2 -9664.287} C_VEL
LIN {X 0,Y 425.284,Z 346.136,A -85,B 0,C 180,E1 -9667.692,E2 -9667.692} C_VEL
LIN {X 0,Y 425.297,Z 346.125,A -85,B 0,C 180,E1 -9670.523,E2 -9670.523} C_VEL
LIN {X 0,Y 425.326,Z 346.129,A -85,B 0,C 180,E1 -9673.36,E2 -9673.36} C_VEL
LIN {X 0,Y 425.325,Z 346.122,A -85,B 0,C 180,E1 -9676.637,E2 -9676.637} C_VEL
LIN {X 0,Y 425.304,Z 346.126,A -85,B 0,C 180,E1 -9679.875,E2 -9679.875} C_VEL
LIN {X 0,Y 425.279,Z 346.11,A -85,B 0,C 180,E1 -9682.486,E2 -9682.486} C_VEL
LIN {X 0,Y 425.299,Z 346.136,A -85,B 0,C 180,E1 -9685.816,E2 -9685.816} C_VEL
LIN {X 0,Y 425.291,Z 346.116,A -85,B 0,C 180,E1 -9689.236,E2 -9689.236} C_VEL
LIN {X 0,Y 425.341,Z 346.107,A -85,B 0,C 180,E1 -9692.442,E2 -9692.442} C_VEL
LIN {X 0,Y 425.345,Z 346.13,A -85,B 0,C 180,E1 -9695.602,E2 -9695.602} C_VEL
LIN {X 0,Y 425.286,Z 346.124,A -85,B 0,C 180,E1 -9698.681,E2 -9698.681} C_VEL
LIN {X 0,Y 425.323,Z 346.129,A -85,B 0,C 180,E1 -9701.702,E2 -9701.702} C_VEL
LIN {X 0,Y 425.338,Z 346.114,A -85,B 0,C 180,E1 -9704.67,E2 -9704.67} C_VEL
LIN {X 0,Y 425.42,Z 346.116,A -85,B 0,C 180,E1 -9707.598,E2 -9707.598} C_VEL
LIN {X 0,Y 425.432,Z 346.11,A -85,B 0,C 180,E1 -9711.45,E2 -9711.45} C_VEL
LIN {X 0,Y 425.547,Z 346.098,A -85,B 0,C 180,E1 -9714.313,E2 -9714.313} C_VEL
LIN {X 0,Y 425.566,Z 346.092,A -85,B 0,C 180,E1 -9718.107,E2 -9718.107} C_VEL
LIN {X 0,Y 425.696,Z 346.081,A -85,B 0,C 180,E1 -9720,E2 -9720} C_VEL
LIN {X 0,Y 425.549,Z 346.092,A -85,B 0,C 180,E1 -9722.84,E2 -9722.84} C_VEL
LIN {X 0,Y 425.522,Z 346.105,A -85,B 0,C 180,E1 -9726.639,E2 -9726.639} C_VEL
LIN {X 0,Y 425.394,Z 346.106,A -85,B 0,C 180,E1 -9729.509,E2 -9729.509} C_VEL
LIN {X 0,Y 425.393,Z 346.12,A -85,B 0,C 180,E1 -9732.911,E2 -9732.911} C_VEL
LIN {X 0,Y 425.35,Z 346.117,A -85,B 0,C 180,E1 -9736.605,E2 -9736.605} C_VEL
LIN {X 0,Y 425.318,Z 346.124,A -85,B 0,C 180,E1 -9739.636,E2 -9739.636} C_VEL
LIN {X 0,Y 425.298,Z 346.13,A -85,B 0,C 180,E1 -9743.366,E2 -9743.366} C_VEL
LIN {X 0,Y 425.339,Z 346.11,A -85,B 0,C 180,E1 -9746.845,E2 -9746.845} C_VEL
LIN {X 0,Y 425.281,Z 346.103,A -85,B 0,C 180,E1 -9749.72,E2 -9749.72} C_VEL
LIN {X 0,Y 425.273,Z 346.135,A -85,B 0,C 180,E1 -9753.049,E2 -9753.049} C_VEL
LIN {X 0,Y 425.276,Z 346.127,A -85,B 0,C 180,E1 -9755.93,E2 -9755.93} C_VEL
LIN {X 0,Y 425.304,Z 346.118,A -85,B 0,C 180,E1 -9759.047,E2 -9759.047} C_VEL
LIN {X 0,Y 425.324,Z 346.125,A -85,B 0,C 180,E1 -9762.647,E2 -9762.647} C_VEL
LIN {X 0,Y 425.327,Z 346.118,A -85,B 0,C 180,E1 -9766.055,E2 -9766.055} C_VEL
LIN {X 0,Y 425.303,Z 346.128,A -85,B 0,C 180,E1 -9768.627,E2 -9768.627} C_VEL
LIN {X 0,Y 425.318,Z 346.125,A -85,B 0,C 180,E1 -9771.105,E2 -9771.105} C_VEL
LIN {X 0,Y 425.295,Z 346.128,A -85,B 0,C 180,E1 -9774.666,E2 -9774.666} C_VEL
LIN {X 0,Y 425.269,Z 346.135,A -85,B 0,C 180,E1 -9778.075,E2 -9778.075} C_VEL
LIN {X 0,Y 425.371,Z 346.133,A -85,B 0,C 180,E1 -9781.776,E2 -9781.776} C_VEL
LIN {X 0,Y 425.408,Z 346.329,A -85,B 0,C 180,E1 -9781.913,E2 -9781.913} C_VEL
LIN {X 0,Y 428.041,Z 358.416,A -85,B 0,C 180,E1 -9784.561,E2 -9784.561} C_VEL
LIN {X 0,Y 429.159,Z 364.498,A -85,B 0,C 180,E1 -9785.834,E2 -9785.834} C_VEL
LIN {X 0,Y 428.595,Z 372.181,A -85,B 0,C 180,E1 -9787.268,E2 -9787.268} C_VEL
LIN {X 0,Y 430.861,Z 383.019,A -85,B 0,C 180,E1 -9787.62,E2 -9787.62} C_VEL
LIN {X 0,Y 433.651,Z 397.443,A -85,B 0,C 180,E1 -9788.024,E2 -9788.024} C_VEL
LIN {X 0,Y 432.273,Z 502.812,A -85,B 0,C 180,E1 -9789.79,E2 -9789.79} C_VEL
LIN {X 0,Y 431.839,Z 517.566,A -85,B 0,C 180,E1 -9790.141,E2 -9790.141} C_VEL
LIN {X 0,Y 431.193,Z 531.623,A -85,B 0,C 180,E1 -9790.668,E2 -9790.668} C_VEL
LIN {X 0,Y 430.489,Z 545.305,A -85,B 0,C 180,E1 -9791.383,E2 -9791.383} C_VEL
LIN {X 0,Y 429.631,Z 558.268,A -85,B 0,C 180,E1 -9792.263,E2 -9792.263} C_VEL
LIN {X 0,Y 428.638,Z 570.757,A -85,B 0,C 180,E1 -9793.327,E2 -9793.327} C_VEL
LIN {X 0,Y 427.688,Z 582.047,A -85,B 0,C 180,E1 -9794.514,E2 -9794.514} C_VEL
LIN {X 0,Y 426.834,Z 591.418,A -85,B 0,C 180,E1 -9795.702,E2 -9795.702} C_VEL
LIN {X 0,Y 426.119,Z 600.921,A -85,B 0,C 180,E1 -9797.149,E2 -9797.149} C_VEL
LIN {X 0,Y 425.357,Z 609.819,A -85,B 0,C 180,E1 -9798.807,E2 -9798.807} C_VEL
LIN {X 0,Y 424.835,Z 617.066,A -85,B 0,C 180,E1 -9800.479,E2 -9800.479} C_VEL
LIN {X 0,Y 424.497,Z 622.144,A -85,B 0,C 180,E1 -9801.911,E2 -9801.911} C_VEL
LIN {X 0,Y 424.33,Z 626.861,A -85,B 0,C 180,E1 -9803.594,E2 -9803.594} C_VEL
LIN {X 0,Y 424.187,Z 630.325,A -85,B 0,C 180,E1 -9805.249,E2 -9805.249} C_VEL
LIN {X 0,Y 424.09,Z 633.009,A -85,B 0,C 180,E1 -9807.152,E2 -9807.152} C_VEL
LIN {X 0,Y 424.067,Z 634.336,A -85,B 0,C 180,E1 -9809.052,E2 -9809.052} C_VEL
LIN {X 0,Y 424.067,Z 634.333,A -85,B 0,C 180,E1 -9810.951,E2 -9810.951} C_VEL
LIN {X 0,Y 424.091,Z 632.999,A -85,B 0,C 180,E1 -9812.851,E2 -9812.851} C_VEL
LIN {X 0,Y 424.187,Z 630.31,A -85,B 0,C 180,E1 -9814.753,E2 -9814.753} C_VEL
LIN {X 0,Y 424.3,Z 626.193,A -85,B 0,C 180,E1 -9816.659,E2 -9816.659} C_VEL
LIN {X 0,Y 424.614,Z 620.517,A -85,B 0,C 180,E1 -9818.568,E2 -9818.568} C_VEL
LIN {X 0,Y 425.036,Z 614.113,A -85,B 0,C 180,E1 -9820.24,E2 -9820.24} C_VEL
LIN {X 0,Y 425.691,Z 606.157,A -85,B 0,C 180,E1 -9821.911,E2 -9821.911} C_VEL
LIN {X 0,Y 426.396,Z 597,A -85,B 0,C 180,E1 -9823.478,E2 -9823.478} C_VEL
LIN {X 0,Y 427.149,Z 587.805,A -85,B 0,C 180,E1 -9824.776,E2 -9824.776} C_VEL
LIN {X 0,Y 428.122,Z 576.618,A -85,B 0,C 180,E1 -9826.083,E2 -9826.083} C_VEL
LIN {X 0,Y 429.045,Z 565.48,A -85,B 0,C 180,E1 -9827.15,E2 -9827.15} C_VEL
LIN {X 0,Y 429.947,Z 553.349,A -85,B 0,C 180,E1 -9828.095,E2 -9828.095} C_VEL
LIN {X 0,Y 430.73,Z 541.207,A -85,B 0,C 180,E1 -9828.852,E2 -9828.852} C_VEL
LIN {X 0,Y 431.379,Z 527.337,A -85,B 0,C 180,E1 -9829.512,E2 -9829.512} C_VEL
LIN {X 0,Y 432.013,Z 513.168,A -85,B 0,C 180,E1 -9829.977,E2 -9829.977} C_VEL
LIN {X 0,Y 432.382,Z 493.454,A -85,B 0,C 180,E1 -9830.362,E2 -9830.362} C_VEL
LIN {X 0,Y 433.684,Z 398.652,A -85,B 0,C 180,E1 -9831.947,E2 -9831.947} C_VEL
LIN {X 0,Y 429.934,Z 378.484,A -85,B 0,C 180,E1 -9832.505,E2 -9832.505} C_VEL
LIN {X 0,Y 428.633,Z 372.175,A -85,B 0,C 180,E1 -9832.728,E2 -9832.728} C_VEL
LIN {X 0,Y 429.129,Z 364.45,A -85,B 0,C 180,E1 -9834.17,E2 -9834.17} C_VEL
LIN {X 0,Y 427.124,Z 353.986,A -85,B 0,C 180,E1 -9836.377,E2 -9836.377} C_VEL
LIN {X 0,Y 425.388,Z 346.292,A -85,B 0,C 180,E1 -9838.091,E2 -9838.091} C_VEL
LIN {X 0,Y 425.292,Z 346.135,A -85,B 0,C 180,E1 -9840.817,E2 -9840.817} C_VEL
LIN {X 0,Y 425.317,Z 346.131,A -85,B 0,C 180,E1 -9844.289,E2 -9844.289} C_VEL
LIN {X 0,Y 425.29,Z 346.134,A -85,B 0,C 180,E1 -9847.694,E2 -9847.694} C_VEL
LIN {X 0,Y 425.284,Z 346.135,A -85,B 0,C 180,E1 -9850.521,E2 -9850.521} C_VEL
LIN {X 0,Y 425.262,Z 346.136,A -85,B 0,C 180,E1 -9853.351,E2 -9853.351} C_VEL
LIN {X 0,Y 425.262,Z 346.137,A -85,B 0,C 180,E1 -9856.65,E2 -9856.65} C_VEL
LIN {X 0,Y 425.291,Z 346.135,A -85,B 0,C 180,E1 -9859.873,E2 -9859.873} C_VEL
LIN {X 0,Y 425.283,Z 346.135,A -85,B 0,C 180,E1 -9862.489,E2 -9862.489} C_VEL
LIN {X 0,Y 425.312,Z 346.133,A -85,B 0,C 180,E1 -9865.818,E2 -9865.818} C_VEL
LIN {X 0,Y 425.309,Z 346.339,A -85,B 0,C 180,E1 -9868.948,E2 -9868.948} C_VEL
LIN {X 0,Y 428.366,Z 356.272,A -85,B 0,C 180,E1 -9870.871,E2 -9870.871} C_VEL
LIN {X 0,Y 430.777,Z 367.314,A -85,B 0,C 180,E1 -9872.818,E2 -9872.818} C_VEL
LIN {X 0,Y 430.748,Z 372.345,A -85,B 0,C 180,E1 -9873.602,E2 -9873.602} C_VEL
LIN {X 0,Y 429.5,Z 395.9,A -85,B 0,C 180,E1 -9877.131,E2 -9877.131} C_VEL
LIN {X 0,Y 428.354,Z 420.644,A -85,B 0,C 180,E1 -9880.797,E2 -9880.797} C_VEL
LIN {X 0,Y 430.981,Z 436.56,A -85,B 0,C 180,E1 -9881.362,E2 -9881.362} C_VEL
LIN {X 0,Y 431.474,Z 443.293,A -85,B 0,C 180,E1 -9881.554,E2 -9881.554} C_VEL
LIN {X 0,Y 429.882,Z 511.652,A -85,B 0,C 180,E1 -9883.039,E2 -9883.039} C_VEL
LIN {X 0,Y 429.392,Z 533.688,A -85,B 0,C 180,E1 -9883.539,E2 -9883.539} C_VEL
LIN {X 0,Y 428.886,Z 546.424,A -85,B 0,C 180,E1 -9884.008,E2 -9884.008} C_VEL
LIN {X 0,Y 428.273,Z 559.016,A -85,B 0,C 180,E1 -9884.656,E2 -9884.656} C_VEL
LIN {X 0,Y 427.632,Z 571.093,A -85,B 0,C 180,E1 -9885.485,E2 -9885.485} C_VEL
LIN {X 0,Y 426.874,Z 583.19,A -85,B 0,C 180,E1 -9886.544,E2 -9886.544} C_VEL
LIN {X 0,Y 426.261,Z 593.027,A -85,B 0,C 180,E1 -9887.623,E2 -9887.623} C_VEL
LIN {X 0,Y 425.638,Z 601.93,A -85,B 0,C 180,E1 -9888.813,E2 -9888.813} C_VEL
LIN {X 0,Y 425.114,Z 610.635,A -85,B 0,C 180,E1 -9890.244,E2 -9890.244} C_VEL
LIN {X 0,Y 424.706,Z 617.581,A -85,B 0,C 180,E1 -9891.675,E2 -9891.675} C_VEL
LIN {X 0,Y 424.389,Z 623.95,A -85,B 0,C 180,E1 -9893.343,E2 -9893.343} C_VEL
LIN {X 0,Y 424.303,Z 628.072,A -85,B 0,C 180,E1 -9894.773,E2 -9894.773} C_VEL
LIN {X 0,Y 424.108,Z 631.098,A -85,B 0,C 180,E1 -9896.199,E2 -9896.199} C_VEL
LIN {X 0,Y 424.112,Z 632.529,A -85,B 0,C 180,E1 -9897.151,E2 -9897.151} C_VEL
LIN {X 0,Y 424.125,Z 633.536,A -85,B 0,C 180,E1 -9898.101,E2 -9898.101} C_VEL
LIN {X 0,Y 424.071,Z 634.136,A -85,B 0,C 180,E1 -9899.05,E2 -9899.05} C_VEL
LIN {X 0,Y 424.043,Z 634.278,A -85,B 0,C 180,E1 -9900,E2 -9900} C_VEL
LIN {X 0,Y 424.071,Z 633.987,A -85,B 0,C 180,E1 -9900.95,E2 -9900.95} C_VEL
LIN {X 0,Y 424.124,Z 633.29,A -85,B 0,C 180,E1 -9901.899,E2 -9901.899} C_VEL
LIN {X 0,Y 424.096,Z 632.154,A -85,B 0,C 180,E1 -9902.85,E2 -9902.85} C_VEL
LIN {X 0,Y 424.147,Z 629.605,A -85,B 0,C 180,E1 -9904.276,E2 -9904.276} C_VEL
LIN {X 0,Y 424.249,Z 625.992,A -85,B 0,C 180,E1 -9905.704,E2 -9905.704} C_VEL
LIN {X 0,Y 424.415,Z 621.214,A -85,B 0,C 180,E1 -9907.134,E2 -9907.134} C_VEL
LIN {X 0,Y 424.677,Z 615.136,A -85,B 0,C 180,E1 -9908.566,E2 -9908.566} C_VEL
LIN {X 0,Y 425.057,Z 607.552,A -85,B 0,C 180,E1 -9909.998,E2 -9909.998} C_VEL
LIN {X 0,Y 425.443,Z 599.767,A -85,B 0,C 180,E1 -9911.192,E2 -9911.192} C_VEL
LIN {X 0,Y 426.055,Z 589.222,A -85,B 0,C 180,E1 -9912.504,E2 -9912.504} C_VEL
LIN {X 0,Y 426.624,Z 578.861,A -85,B 0,C 180,E1 -9913.546,E2 -9913.546} C_VEL
LIN {X 0,Y 427.202,Z 566.473,A -85,B 0,C 180,E1 -9914.53,E2 -9914.53} C_VEL
LIN {X 0,Y 427.818,Z 553.818,A -85,B 0,C 180,E1 -9915.3,E2 -9915.3} C_VEL
LIN {X 0,Y 428.292,Z 539.587,A -85,B 0,C 180,E1 -9915.923,E2 -9915.923} C_VEL
LIN {X 0,Y 428.713,Z 525.768,A -85,B 0,C 180,E1 -9916.304,E2 -9916.304} C_VEL
LIN {X 0,Y 429.967,Z 440.427,A -85,B 0,C 180,E1 -9917.99,E2 -9917.99} C_VEL
LIN {X 0,Y 427.263,Z 420.727,A -85,B 0,C 180,E1 -9918.519,E2 -9918.519} C_VEL
LIN {X 0,Y 428.068,Z 401.217,A -85,B 0,C 180,E1 -9921.426,E2 -9921.426} C_VEL
LIN {X 0,Y 429.069,Z 379.516,A -85,B 0,C 180,E1 -9924.688,E2 -9924.688} C_VEL
LIN {X 0,Y 429.594,Z 365.983,A -85,B 0,C 180,E1 -9926.737,E2 -9926.737} C_VEL
LIN {X 0,Y 427.461,Z 355.426,A -85,B 0,C 180,E1 -9928.477,E2 -9928.477} C_VEL
LIN {X 0,Y 425.338,Z 346.257,A -85,B 0,C 180,E1 -9930.057,E2 -9930.057} C_VEL
LIN {X 0,Y 425.288,Z 346.135,A -85,B 0,C 180,E1 -9933.048,E2 -9933.048} C_VEL
LIN {X 0,Y 425.288,Z 346.135,A -85,B 0,C 180,E1 -9935.928,E2 -9935.928} C_VEL
LIN {X 0,Y 425.286,Z 346.132,A -85,B 0,C 180,E1 -9939.04,E2 -9939.04} C_VEL
LIN {X 0,Y 425.295,Z 346.135,A -85,B 0,C 180,E1 -9941.958,E2 -9941.958} C_VEL
LIN {X 0,Y 425.29,Z 346.116,A -85,B 0,C 180,E1 -9945.283,E2 -9945.283} C_VEL
LIN {X 0,Y 425.28,Z 346.132,A -85,B 0,C 180,E1 -9948.621,E2 -9948.621} C_VEL
LIN {X 0,Y 425.318,Z 346.124,A -85,B 0,C 180,E1 -9951.102,E2 -9951.102} C_VEL
LIN {X 0,Y 425.306,Z 346.126,A -85,B 0,C 180,E1 -9954.664,E2 -9954.664} C_VEL
LIN {X 0,Y 425.27,Z 346.134,A -85,B 0,C 180,E1 -9958.072,E2 -9958.072} C_VEL
LIN {X 0,Y 425.387,Z 346.145,A -85,B 0,C 180,E1 -9961.875,E2 -9961.875} C_VEL
LIN {X 0,Y 425.612,Z 347.227,A -85,B 0,C 180,E1 -9962.193,E2 -9962.193} C_VEL
LIN {X 0,Y 428.428,Z 360.299,A -85,B 0,C 180,E1 -9965.012,E2 -9965.012} C_VEL
LIN {X 0,Y 429.149,Z 365.411,A -85,B 0,C 180,E1 -9966.065,E2 -9966.065} C_VEL
LIN {X 0,Y 428.624,Z 372.304,A -85,B 0,C 180,E1 -9967.331,E2 -9967.331} C_VEL
LIN {X 0,Y 433.574,Z 397.007,A -85,B 0,C 180,E1 -9968.063,E2 -9968.063} C_VEL
LIN {X 0,Y 433.244,Z 432.116,A -85,B 0,C 180,E1 -9968.659,E2 -9968.659} C_VEL
LIN {X 0,Y 432.596,Z 437.96,A -85,B 0,C 180,E1 -9968.728,E2 -9968.728} C_VEL
LIN {X 0,Y 426.941,Z 456.979,A -85,B 0,C 180,E1 -9968.768,E2 -9968.768} C_VEL
LIN {X 0,Y 426.251,Z 462.826,A -85,B 0,C 180,E1 -9968.836,E2 -9968.836} C_VEL
LIN {X 0,Y 425.436,Z 510.389,A -85,B 0,C 180,E1 -9969.669,E2 -9969.669} C_VEL
LIN {X 0,Y 424.802,Z 524.716,A -85,B 0,C 180,E1 -9970.11,E2 -9970.11} C_VEL
LIN {X 0,Y 424.149,Z 538.98,A -85,B 0,C 180,E1 -9970.766,E2 -9970.766} C_VEL
LIN {X 0,Y 423.234,Z 552.711,A -85,B 0,C 180,E1 -9971.608,E2 -9971.608} C_VEL
LIN {X 0,Y 422.311,Z 564.964,A -85,B 0,C 180,E1 -9972.568,E2 -9972.568} C_VEL
LIN {X 0,Y 421.309,Z 576.192,A -85,B 0,C 180,E1 -9973.649,E2 -9973.649} C_VEL
LIN {X 0,Y 420.315,Z 587.478,A -85,B 0,C 180,E1 -9974.978,E2 -9974.978} C_VEL
LIN {X 0,Y 419.373,Z 597.559,A -85,B 0,C 180,E1 -9976.43,E2 -9976.43} C_VEL
LIN {X 0,Y 418.735,Z 605.93,A -85,B 0,C 180,E1 -9977.888,E2 -9977.888} C_VEL
LIN {X 0,Y 418.034,Z 613.926,A -85,B 0,C 180,E1 -9979.587,E2 -9979.587} C_VEL
LIN {X 0,Y 417.561,Z 620.367,A -85,B 0,C 180,E1 -9981.286,E2 -9981.286} C_VEL
LIN {X 0,Y 417.233,Z 626.077,A -85,B 0,C 180,E1 -9983.227,E2 -9983.227} C_VEL
LIN {X 0,Y 417.118,Z 630.226,A -85,B 0,C 180,E1 -9985.166,E2 -9985.166} C_VEL
LIN {X 0,Y 416.99,Z 632.946,A -85,B 0,C 180,E1 -9987.101,E2 -9987.101} C_VEL
LIN {X 0,Y 416.991,Z 634.312,A -85,B 0,C 180,E1 -9989.033,E2 -9989.033} C_VEL
LIN {X 0,Y 416.991,Z 634.351,A -85,B 0,C 180,E1 -9990.964,E2 -9990.964} C_VEL
LIN {X 0,Y 416.989,Z 633.061,A -85,B 0,C 180,E1 -9992.897,E2 -9992.897} C_VEL
LIN {X 0,Y 417.117,Z 630.409,A -85,B 0,C 180,E1 -9994.831,E2 -9994.831} C_VEL
LIN {X 0,Y 417.231,Z 626.325,A -85,B 0,C 180,E1 -9996.77,E2 -9996.77} C_VEL
LIN {X 0,Y 417.548,Z 620.687,A -85,B 0,C 180,E1 -9998.712,E2 -9998.712} C_VEL
LIN {X 0,Y 417.986,Z 614.327,A -85,B 0,C 180,E1 -10000.412,E2 -10000.412} C_VEL
LIN {X 0,Y 418.692,Z 606.418,A -85,B 0,C 180,E1 -10002.11,E2 -10002.11} C_VEL
LIN {X 0,Y 419.371,Z 597.996,A -85,B 0,C 180,E1 -10003.593,E2 -10003.593} C_VEL
LIN {X 0,Y 420.231,Z 588.182,A -85,B 0,C 180,E1 -10005.023,E2 -10005.023} C_VEL
LIN {X 0,Y 421.252,Z 577.093,A -85,B 0,C 180,E1 -10006.35,E2 -10006.35} C_VEL
LIN {X 0,Y 422.346,Z 564.66,A -85,B 0,C 180,E1 -10007.553,E2 -10007.553} C_VEL
LIN {X 0,Y 423.307,Z 552.237,A -85,B 0,C 180,E1 -10008.519,E2 -10008.519} C_VEL
LIN {X 0,Y 424.154,Z 538.58,A -85,B 0,C 180,E1 -10009.352,E2 -10009.352} C_VEL
LIN {X 0,Y 424.87,Z 524.801,A -85,B 0,C 180,E1 -10009.978,E2 -10009.978} C_VEL
LIN {X 0,Y 425.471,Z 510.529,A -85,B 0,C 180,E1 -10010.421,E2 -10010.421} C_VEL
LIN {X 0,Y 426.155,Z 467.851,A -85,B 0,C 180,E1 -10011.177,E2 -10011.177} C_VEL
LIN {X 0,Y 426.98,Z 397.787,A -85,B 0,C 180,E1 -10012.377,E2 -10012.377} C_VEL
LIN {X 0,Y 421.866,Z 372.503,A -85,B 0,C 180,E1 -10013.14,E2 -10013.14} C_VEL
LIN {X 0,Y 421.988,Z 369.486,A -85,B 0,C 180,E1 -10013.652,E2 -10013.652} C_VEL
LIN {X 0,Y 422.282,Z 366.163,A -85,B 0,C 180,E1 -10014.297,E2 -10014.297} C_VEL
LIN {X 0,Y 419.989,Z 354.26,A -85,B 0,C 180,E1 -10016.858,E2 -10016.858} C_VEL
LIN {X 0,Y 418.364,Z 347.205,A -85,B 0,C 180,E1 -10018.466,E2 -10018.466} C_VEL
LIN {X 0,Y 418.22,Z 347.016,A -85,B 0,C 180,E1 -10021.394,E2 -10021.394} C_VEL
LIN {X 0,Y 418.262,Z 347.009,A -85,B 0,C 180,E1 -10024.579,E2 -10024.579} C_VEL
LIN {X 0,Y 418.234,Z 347.016,A -85,B 0,C 180,E1 -10027.834,E2 -10027.834} C_VEL
LIN {X 0,Y 418.262,Z 347.003,A -85,B 0,C 180,E1 -10030.941,E2 -10030.941} C_VEL
LIN {X 0,Y 418.277,Z 347,A -85,B 0,C 180,E1 -10033.739,E2 -10033.739} C_VEL
LIN {X 0,Y 418.276,Z 346.999,A -85,B 0,C 180,E1 -10036.457,E2 -10036.457} C_VEL
LIN {X 0,Y 418.26,Z 347.008,A -85,B 0,C 180,E1 -10039.122,E2 -10039.122} C_VEL
LIN {X 0,Y 418.23,Z 346.986,A -85,B 0,C 180,E1 -10042.164,E2 -10042.164} C_VEL
LIN {X 0,Y 418.257,Z 347.008,A -85,B 0,C 180,E1 -10045.419,E2 -10045.419} C_VEL
LIN {X 0,Y 418.208,Z 347.005,A -85,B 0,C 180,E1 -10048.603,E2 -10048.603} C_VEL
LIN {X 0,Y 418.286,Z 346.976,A -85,B 0,C 180,E1 -10051.936,E2 -10051.936} C_VEL
LIN {X 0,Y 418.28,Z 347.004,A -85,B 0,C 180,E1 -10055.162,E2 -10055.162} C_VEL
LIN {X 0,Y 418.226,Z 347.003,A -85,B 0,C 180,E1 -10058.303,E2 -10058.303} C_VEL
LIN {X 0,Y 418.274,Z 347.01,A -85,B 0,C 180,E1 -10061.383,E2 -10061.383} C_VEL
LIN {X 0,Y 418.292,Z 346.991,A -85,B 0,C 180,E1 -10064.405,E2 -10064.405} C_VEL
LIN {X 0,Y 418.36,Z 346.998,A -85,B 0,C 180,E1 -10067.386,E2 -10067.386} C_VEL
LIN {X 0,Y 418.351,Z 346.983,A -85,B 0,C 180,E1 -10070.329,E2 -10070.329} C_VEL
LIN {X 0,Y 418.484,Z 346.984,A -85,B 0,C 180,E1 -10073.249,E2 -10073.249} C_VEL
LIN {X 0,Y 418.335,Z 346.995,A -85,B 0,C 180,E1 -10075.181,E2 -10075.181} C_VEL
LIN {X 0,Y 418.535,Z 346.967,A -85,B 0,C 180,E1 -10078.075,E2 -10078.075} C_VEL
LIN {X 0,Y 418.665,Z 346.956,A -85,B 0,C 180,E1 -10080,E2 -10080} C_VEL
LIN {X 0,Y 418.503,Z 346.969,A -85,B 0,C 180,E1 -10082.888,E2 -10082.888} C_VEL
LIN {X 0,Y 418.484,Z 346.983,A -85,B 0,C 180,E1 -10086.751,E2 -10086.751} C_VEL
LIN {X 0,Y 418.35,Z 346.983,A -85,B 0,C 180,E1 -10089.671,E2 -10089.671} C_VEL
LIN {X 0,Y 418.344,Z 346.996,A -85,B 0,C 180,E1 -10093.007,E2 -10093.007} C_VEL
LIN {X 0,Y 418.302,Z 346.996,A -85,B 0,C 180,E1 -10096.736,E2 -10096.736} C_VEL
LIN {X 0,Y 418.261,Z 347.003,A -85,B 0,C 180,E1 -10099.791,E2 -10099.791} C_VEL
LIN {X 0,Y 418.228,Z 347.011,A -85,B 0,C 180,E1 -10102.737,E2 -10102.737} C_VEL
LIN {X 0,Y 418.264,Z 347.004,A -85,B 0,C 180,E1 -10105.904,E2 -10105.904} C_VEL
LIN {X 0,Y 418.255,Z 346.974,A -85,B 0,C 180,E1 -10109.163,E2 -10109.163} C_VEL
LIN {X 0,Y 418.248,Z 347.011,A -85,B 0,C 180,E1 -10112.845,E2 -10112.845} C_VEL
LIN {X 0,Y 418.24,Z 346.996,A -85,B 0,C 180,E1 -10116.24,E2 -10116.24} C_VEL
LIN {X 0,Y 418.258,Z 346.998,A -85,B 0,C 180,E1 -10119.681,E2 -10119.681} C_VEL
LIN {X 0,Y 418.277,Z 347.006,A -85,B 0,C 180,E1 -10122.331,E2 -10122.331} C_VEL
LIN {X 0,Y 418.267,Z 346.99,A -85,B 0,C 180,E1 -10125.115,E2 -10125.115} C_VEL
LIN {X 0,Y 418.286,Z 347.008,A -85,B 0,C 180,E1 -10127.775,E2 -10127.775} C_VEL
LIN {X 0,Y 418.261,Z 347.006,A -85,B 0,C 180,E1 -10131.561,E2 -10131.561} C_VEL
LIN {X 0,Y 418.255,Z 347.008,A -85,B 0,C 180,E1 -10135.16,E2 -10135.16} C_VEL
LIN {X 0,Y 418.245,Z 347.005,A -85,B 0,C 180,E1 -10137.474,E2 -10137.474} C_VEL
LIN {X 0,Y 418.273,Z 346.982,A -85,B 0,C 180,E1 -10140.895,E2 -10140.895} C_VEL
LIN {X 0,Y 418.328,Z 347.099,A -85,B 0,C 180,E1 -10141.531,E2 -10141.531} C_VEL
LIN {X 0,Y 420.48,Z 356.656,A -85,B 0,C 180,E1 -10143.711,E2 -10143.711} C_VEL
LIN {X 0,Y 422.248,Z 365.809,A -85,B 0,C 180,E1 -10145.675,E2 -10145.675} C_VEL
LIN {X 0,Y 421.794,Z 372.181,A -85,B 0,C 180,E1 -10146.88,E2 -10146.88} C_VEL
LIN {X 0,Y 424.184,Z 383.465,A -85,B 0,C 180,E1 -10147.256,E2 -10147.256} C_VEL
LIN {X 0,Y 427.11,Z 399.173,A -85,B 0,C 180,E1 -10147.7,E2 -10147.7} C_VEL
LIN {X 0,Y 425.59,Z 504.333,A -85,B 0,C 180,E1 -10149.49,E2 -10149.49} C_VEL
LIN {X 0,Y 425.152,Z 518.49,A -85,B 0,C 180,E1 -10149.847,E2 -10149.847} C_VEL
LIN {X 0,Y 424.44,Z 532.93,A -85,B 0,C 180,E1 -10150.41,E2 -10150.41} C_VEL
LIN {X 0,Y 423.697,Z 546.273,A -85,B 0,C 180,E1 -10151.134,E2 -10151.134} C_VEL
LIN {X 0,Y 422.848,Z 558.273,A -85,B 0,C 180,E1 -10151.969,E2 -10151.969} C_VEL
LIN {X 0,Y 421.821,Z 570.76,A -85,B 0,C 180,E1 -10153.049,E2 -10153.049} C_VEL
LIN {X 0,Y 420.808,Z 582.049,A -85,B 0,C 180,E1 -10154.254,E2 -10154.254} C_VEL
LIN {X 0,Y 419.915,Z 591.421,A -85,B 0,C 180,E1 -10155.462,E2 -10155.462} C_VEL
LIN {X 0,Y 419.122,Z 601.188,A -85,B 0,C 180,E1 -10156.977,E2 -10156.977} C_VEL
LIN {X 0,Y 418.38,Z 609.82,A -85,B 0,C 180,E1 -10158.618,E2 -10158.618} C_VEL
LIN {X 0,Y 417.798,Z 617.067,A -85,B 0,C 180,E1 -10160.317,E2 -10160.317} C_VEL
LIN {X 0,Y 417.338,Z 623.578,A -85,B 0,C 180,E1 -10162.259,E2 -10162.259} C_VEL
LIN {X 0,Y 417.26,Z 627.114,A -85,B 0,C 180,E1 -10163.591,E2 -10163.591} C_VEL
LIN {X 0,Y 417.118,Z 630.326,A -85,B 0,C 180,E1 -10165.169,E2 -10165.169} C_VEL
LIN {X 0,Y 416.989,Z 633.009,A -85,B 0,C 180,E1 -10167.103,E2 -10167.103} C_VEL
LIN {X 0,Y 416.99,Z 634.336,A -85,B 0,C 180,E1 -10169.036,E2 -10169.036} C_VEL
LIN {X 0,Y 416.99,Z 634.333,A -85,B 0,C 180,E1 -10170.967,E2 -10170.967} C_VEL
LIN {X 0,Y 416.989,Z 632.998,A -85,B 0,C 180,E1 -10172.899,E2 -10172.899} C_VEL
LIN {X 0,Y 417.117,Z 630.309,A -85,B 0,C 180,E1 -10174.834,E2 -10174.834} C_VEL
LIN {X 0,Y 417.231,Z 626.192,A -85,B 0,C 180,E1 -10176.773,E2 -10176.773} C_VEL
LIN {X 0,Y 417.551,Z 620.516,A -85,B 0,C 180,E1 -10178.714,E2 -10178.714} C_VEL
LIN {X 0,Y 418.002,Z 614.112,A -85,B 0,C 180,E1 -10180.414,E2 -10180.414} C_VEL
LIN {X 0,Y 418.713,Z 606.155,A -85,B 0,C 180,E1 -10182.112,E2 -10182.112} C_VEL
LIN {X 0,Y 419.416,Z 597.529,A -85,B 0,C 180,E1 -10183.619,E2 -10183.619} C_VEL
LIN {X 0,Y 420.257,Z 587.803,A -85,B 0,C 180,E1 -10185.024,E2 -10185.024} C_VEL
LIN {X 0,Y 421.262,Z 576.615,A -85,B 0,C 180,E1 -10186.353,E2 -10186.353} C_VEL
LIN {X 0,Y 422.38,Z 564.051,A -85,B 0,C 180,E1 -10187.554,E2 -10187.554} C_VEL
LIN {X 0,Y 423.313,Z 551.436,A -85,B 0,C 180,E1 -10188.524,E2 -10188.524} C_VEL
LIN {X 0,Y 424.235,Z 537.631,A -85,B 0,C 180,E1 -10189.35,E2 -10189.35} C_VEL
LIN {X 0,Y 424.875,Z 524.28,A -85,B 0,C 180,E1 -10189.949,E2 -10189.949} C_VEL
LIN {X 0,Y 425.436,Z 509.735,A -85,B 0,C 180,E1 -10190.394,E2 -10190.394} C_VEL
LIN {X 0,Y 426.818,Z 420.123,A -85,B 0,C 180,E1 -10191.937,E2 -10191.937} C_VEL
LIN {X 0,Y 426.956,Z 397.886,A -85,B 0,C 180,E1 -10192.325,E2 -10192.325} C_VEL
LIN {X 0,Y 421.88,Z 372.421,A -85,B 0,C 180,E1 -10193.093,E2 -10193.093} C_VEL
LIN {X 0,Y 422.093,Z 368.503,A -85,B 0,C 180,E1 -10193.789,E2 -10193.789} C_VEL
LIN {X 0,Y 422.23,Z 365.757,A -85,B 0,C 180,E1 -10194.329,E2 -10194.329} C_VEL
LIN {X 0,Y 419.884,Z 353.984,A -85,B 0,C 180,E1 -10196.868,E2 -10196.868} C_VEL
LIN {X 0,Y 418.331,Z 347.067,A -85,B 0,C 180,E1 -10198.471,E2 -10198.471} C_VEL
LIN {X 0,Y 418.216,Z 347.015,A -85,B 0,C 180,E1 -10201.397,E2 -10201.397} C_VEL
LIN {X 0,Y 418.271,Z 347.008,A -85,B 0,C 180,E1 -10204.581,E2 -10204.581} C_VEL
LIN {X 0,Y 418.238,Z 347.012,A -85,B 0,C 180,E1 -10207.835,E2 -10207.835} C_VEL
LIN {X 0,Y 418.226,Z 347.012,A -85,B 0,C 180,E1 -10210.949,E2 -10210.949} C_VEL
LIN {X 0,Y 418.214,Z 347.017,A -85,B 0,C 180,E1 -10213.73,E2 -10213.73} C_VEL
LIN {X 0,Y 418.213,Z 347.015,A -85,B 0,C 180,E1 -10216.449,E2 -10216.449} C_VEL
LIN {X 0,Y 418.228,Z 347.015,A -85,B 0,C 180,E1 -10219.131,E2 -10219.131} C_VEL
LIN {X 0,Y 418.233,Z 347.013,A -85,B 0,C 180,E1 -10222.167,E2 -10222.167} C_VEL
LIN {X 0,Y 418.27,Z 347.011,A -85,B 0,C 180,E1 -10225.42,E2 -10225.42} C_VEL
LIN {X 0,Y 418.261,Z 347.161,A -85,B 0,C 180,E1 -10228.29,E2 -10228.29} C_VEL
LIN {X 0,Y 421.759,Z 358.286,A -85,B 0,C 180,E1 -10230.55,E2 -10230.55} C_VEL
LIN {X 0,Y 423.97,Z 368.102,A -85,B 0,C 180,E1 -10232.345,E2 -10232.345} C_VEL
LIN {X 0,Y 424.371,Z 371.404,A -85,B 0,C 180,E1 -10232.908,E2 -10232.908} C_VEL
LIN {X 0,Y 422.903,Z 396.655,A -85,B 0,C 180,E1 -10236.753,E2 -10236.753} C_VEL
LIN {X 0,Y 421.677,Z 420.476,A -85,B 0,C 180,E1 -10240.339,E2 -10240.339} C_VEL
LIN {X 0,Y 424.25,Z 435.332,A -85,B 0,C 180,E1 -10240.915,E2 -10240.915} C_VEL
LIN {X 0,Y 425.013,Z 443.298,A -85,B 0,C 180,E1 -10241.164,E2 -10241.164} C_VEL
LIN {X 0,Y 423.152,Z 513.168,A -85,B 0,C 180,E1 -10242.73,E2 -10242.73} C_VEL
LIN {X 0,Y 422.693,Z 534.419,A -85,B 0,C 180,E1 -10243.24,E2 -10243.24} C_VEL
LIN {X 0,Y 422.14,Z 547.518,A -85,B 0,C 180,E1 -10243.746,E2 -10243.746} C_VEL
LIN {X 0,Y 421.475,Z 559.782,A -85,B 0,C 180,E1 -10244.402,E2 -10244.402} C_VEL
LIN {X 0,Y 420.798,Z 571.634,A -85,B 0,C 180,E1 -10245.244,E2 -10245.244} C_VEL
LIN {X 0,Y 420.038,Z 582.861,A -85,B 0,C 180,E1 -10246.244,E2 -10246.244} C_VEL
LIN {X 0,Y 419.351,Z 593.349,A -85,B 0,C 180,E1 -10247.416,E2 -10247.416} C_VEL
LIN {X 0,Y 418.681,Z 602.193,A -85,B 0,C 180,E1 -10248.625,E2 -10248.625} C_VEL
LIN {X 0,Y 418.127,Z 610.842,A -85,B 0,C 180,E1 -10250.079,E2 -10250.079} C_VEL
LIN {X 0,Y 417.687,Z 617.748,A -85,B 0,C 180,E1 -10251.534,E2 -10251.534} C_VEL
LIN {X 0,Y 417.319,Z 624.083,A -85,B 0,C 180,E1 -10253.23,E2 -10253.23} C_VEL
LIN {X 0,Y 417.218,Z 628.17,A -85,B 0,C 180,E1 -10254.684,E2 -10254.684} C_VEL
LIN {X 0,Y 417.024,Z 631.168,A -85,B 0,C 180,E1 -10256.135,E2 -10256.135} C_VEL
LIN {X 0,Y 417.011,Z 632.574,A -85,B 0,C 180,E1 -10257.102,E2 -10257.102} C_VEL
LIN {X 0,Y 417.034,Z 633.566,A -85,B 0,C 180,E1 -10258.069,E2 -10258.069} C_VEL
LIN {X 0,Y 416.994,Z 634.145,A -85,B 0,C 180,E1 -10259.034,E2 -10259.034} C_VEL
LIN {X 0,Y 416.965,Z 634.254,A -85,B 0,C 180,E1 -10260,E2 -10260} C_VEL
LIN {X 0,Y 416.994,Z 633.944,A -85,B 0,C 180,E1 -10260.966,E2 -10260.966} C_VEL
LIN {X 0,Y 417.033,Z 633.226,A -85,B 0,C 180,E1 -10261.932,E2 -10261.932} C_VEL
LIN {X 0,Y 416.995,Z 632.047,A -85,B 0,C 180,E1 -10262.898,E2 -10262.898} C_VEL
LIN {X 0,Y 417.075,Z 629.448,A -85,B 0,C 180,E1 -10264.349,E2 -10264.349} C_VEL
LIN {X 0,Y 417.159,Z 625.776,A -85,B 0,C 180,E1 -10265.802,E2 -10265.802} C_VEL
LIN {X 0,Y 417.352,Z 620.931,A -85,B 0,C 180,E1 -10267.256,E2 -10267.256} C_VEL
LIN {X 0,Y 417.612,Z 614.776,A -85,B 0,C 180,E1 -10268.712,E2 -10268.712} C_VEL
LIN {X 0,Y 418,Z 607.088,A -85,B 0,C 180,E1 -10270.168,E2 -10270.168} C_VEL
LIN {X 0,Y 418.546,Z 597.406,A -85,B 0,C 180,E1 -10271.625,E2 -10271.625} C_VEL
LIN {X 0,Y 419.152,Z 587.421,A -85,B 0,C 180,E1 -10272.836,E2 -10272.836} C_VEL
LIN {X 0,Y 419.767,Z 576.214,A -85,B 0,C 180,E1 -10273.926,E2 -10273.926} C_VEL
LIN {X 0,Y 420.281,Z 565.341,A -85,B 0,C 180,E1 -10274.774,E2 -10274.774} C_VEL
LIN {X 0,Y 420.849,Z 553.416,A -85,B 0,C 180,E1 -10275.497,E2 -10275.497} C_VEL
LIN {X 0,Y 421.328,Z 539.882,A -85,B 0,C 180,E1 -10276.1,E2 -10276.1} C_VEL
LIN {X 0,Y 421.772,Z 526.392,A -85,B 0,C 180,E1 -10276.487,E2 -10276.487} C_VEL
LIN {X 0,Y 423.083,Z 441.169,A -85,B 0,C 180,E1 -10278.22,E2 -10278.22} C_VEL
LIN {X 0,Y 420.334,Z 420.766,A -85,B 0,C 180,E1 -10278.776,E2 -10278.776} C_VEL
LIN {X 0,Y 421.28,Z 398.999,A -85,B 0,C 180,E1 -10282.046,E2 -10282.046} C_VEL
LIN {X 0,Y 422.263,Z 378.819,A -85,B 0,C 180,E1 -10285.114,E2 -10285.114} C_VEL
LIN {X 0,Y 422.762,Z 368.635,A -85,B 0,C 180,E1 -10286.67,E2 -10286.67} C_VEL
LIN {X 0,Y 421.983,Z 363.386,A -85,B 0,C 180,E1 -10287.527,E2 -10287.527} C_VEL
LIN {X 0,Y 418.32,Z 347.176,A -85,B 0,C 180,E1 -10290.297,E2 -10290.297} C_VEL
LIN {X 0,Y 418.254,Z 347.011,A -85,B 0,C 180,E1 -10293.677,E2 -10293.677} C_VEL
LIN {X 0,Y 418.245,Z 347.01,A -85,B 0,C 180,E1 -10297.224,E2 -10297.224} C_VEL
LIN {X 0,Y 418.25,Z 347.01,A -85,B 0,C 180,E1 -10299.682,E2 -10299.682} C_VEL
LIN {X 0,Y 418.235,Z 347.012,A -85,B 0,C 180,E1 -10302.321,E2 -10302.321} C_VEL
LIN {X 0,Y 418.241,Z 346.992,A -85,B 0,C 180,E1 -10305.108,E2 -10305.108} C_VEL
LIN {X 0,Y 418.246,Z 347.013,A -85,B 0,C 180,E1 -10307.766,E2 -10307.766} C_VEL
LIN {X 0,Y 418.264,Z 347.005,A -85,B 0,C 180,E1 -10311.558,E2 -10311.558} C_VEL
LIN {X 0,Y 418.265,Z 347.006,A -85,B 0,C 180,E1 -10315.158,E2 -10315.158} C_VEL
LIN {X 0,Y 418.251,Z 347.004,A -85,B 0,C 180,E1 -10317.471,E2 -10317.471} C_VEL
LIN {X 0,Y 418.274,Z 346.982,A -85,B 0,C 180,E1 -10320.895,E2 -10320.895} C_VEL
LIN {X 0,Y 418.358,Z 347.117,A -85,B 0,C 180,E1 -10321.599,E2 -10321.599} C_VEL
LIN {X 0,Y 421.046,Z 359.285,A -85,B 0,C 180,E1 -10324.337,E2 -10324.337} C_VEL
LIN {X 0,Y 422.189,Z 365.532,A -85,B 0,C 180,E1 -10325.668,E2 -10325.668} C_VEL
LIN {X 0,Y 421.841,Z 372.149,A -85,B 0,C 180,E1 -10326.929,E2 -10326.929} C_VEL
LIN {X 0,Y 423.213,Z 378.753,A -85,B 0,C 180,E1 -10327.168,E2 -10327.168} C_VEL
LIN {X 0,Y 427.007,Z 398.068,A -85,B 0,C 180,E1 -10327.726,E2 -10327.726} C_VEL
LIN {X 0,Y 426.251,Z 462.826,A -85,B 0,C 180,E1 -10328.836,E2 -10328.836} C_VEL
LIN {X 0,Y 425.57,Z 468.669,A -85,B 0,C 180,E1 -10328.904,E2 -10328.904} C_VEL
LIN {X 0,Y 419.885,Z 487.675,A -85,B 0,C 180,E1 -10328.945,E2 -10328.945} C_VEL
LIN {X 0,Y 419.155,Z 493.521,A -85,B 0,C 180,E1 -10329.012,E2 -10329.012} C_VEL
LIN {X 0,Y 418.691,Z 512.687,A -85,B 0,C 180,E1 -10329.391,E2 -10329.391} C_VEL
LIN {X 0,Y 418.049,Z 527.013,A -85,B 0,C 180,E1 -10329.872,E2 -10329.872} C_VEL
LIN {X 0,Y 417.321,Z 541.422,A -85,B 0,C 180,E1 -10330.576,E2 -10330.576} C_VEL
LIN {X 0,Y 416.359,Z 554.44,A -85,B 0,C 180,E1 -10331.42,E2 -10331.42} C_VEL
LIN {X 0,Y 415.431,Z 566.341,A -85,B 0,C 180,E1 -10332.397,E2 -10332.397} C_VEL
LIN {X 0,Y 414.378,Z 577.329,A -85,B 0,C 180,E1 -10333.495,E2 -10333.495} C_VEL
LIN {X 0,Y 413.418,Z 587.481,A -85,B 0,C 180,E1 -10334.721,E2 -10334.721} C_VEL
LIN {X 0,Y 412.386,Z 597.986,A -85,B 0,C 180,E1 -10336.267,E2 -10336.267} C_VEL
LIN {X 0,Y 411.641,Z 607.163,A -85,B 0,C 180,E1 -10337.927,E2 -10337.927} C_VEL
LIN {X 0,Y 410.97,Z 614.935,A -85,B 0,C 180,E1 -10339.655,E2 -10339.655} C_VEL
LIN {X 0,Y 410.513,Z 620.369,A -85,B 0,C 180,E1 -10341.135,E2 -10341.135} C_VEL
LIN {X 0,Y 410.165,Z 626.078,A -85,B 0,C 180,E1 -10343.11,E2 -10343.11} C_VEL
LIN {X 0,Y 410.028,Z 630.227,A -85,B 0,C 180,E1 -10345.082,E2 -10345.082} C_VEL
LIN {X 0,Y 409.889,Z 632.947,A -85,B 0,C 180,E1 -10347.05,E2 -10347.05} C_VEL
LIN {X 0,Y 409.917,Z 634.313,A -85,B 0,C 180,E1 -10349.016,E2 -10349.016} C_VEL
LIN {X 0,Y 409.917,Z 634.351,A -85,B 0,C 180,E1 -10350.981,E2 -10350.981} C_VEL
LIN {X 0,Y 409.888,Z 633.06,A -85,B 0,C 180,E1 -10352.947,E2 -10352.947} C_VEL
LIN {X 0,Y 410.026,Z 630.408,A -85,B 0,C 180,E1 -10354.915,E2 -10354.915} C_VEL
LIN {X 0,Y 410.163,Z 626.324,A -85,B 0,C 180,E1 -10356.887,E2 -10356.887} C_VEL
LIN {X 0,Y 410.499,Z 620.685,A -85,B 0,C 180,E1 -10358.862,E2 -10358.862} C_VEL
LIN {X 0,Y 410.964,Z 614.325,A -85,B 0,C 180,E1 -10360.592,E2 -10360.592} C_VEL
LIN {X 0,Y 411.724,Z 606.415,A -85,B 0,C 180,E1 -10362.319,E2 -10362.319} C_VEL
LIN {X 0,Y 412.415,Z 598.143,A -85,B 0,C 180,E1 -10363.801,E2 -10363.801} C_VEL
LIN {X 0,Y 413.354,Z 588.179,A -85,B 0,C 180,E1 -10365.279,E2 -10365.279} C_VEL
LIN {X 0,Y 414.403,Z 577.089,A -85,B 0,C 180,E1 -10366.628,E2 -10366.628} C_VEL
LIN {X 0,Y 415.548,Z 564.655,A -85,B 0,C 180,E1 -10367.849,E2 -10367.849} C_VEL
LIN {X 0,Y 416.563,Z 552.429,A -85,B 0,C 180,E1 -10368.815,E2 -10368.815} C_VEL
LIN {X 0,Y 417.458,Z 538.572,A -85,B 0,C 180,E1 -10369.675,E2 -10369.675} C_VEL
LIN {X 0,Y 418.207,Z 524.79,A -85,B 0,C 180,E1 -10370.31,E2 -10370.31} C_VEL
LIN {X 0,Y 418.835,Z 510.512,A -85,B 0,C 180,E1 -10370.76,E2 -10370.76} C_VEL
LIN {X 0,Y 419.591,Z 466.036,A -85,B 0,C 180,E1 -10371.557,E2 -10371.557} C_VEL
LIN {X 0,Y 420.497,Z 399.219,A -85,B 0,C 180,E1 -10372.714,E2 -10372.714} C_VEL
LIN {X 0,Y 415.189,Z 373.268,A -85,B 0,C 180,E1 -10373.506,E2 -10373.506} C_VEL
LIN {X 0,Y 415.014,Z 371.927,A -85,B 0,C 180,E1 -10373.599,E2 -10373.599} C_VEL
LIN {X 0,Y 415.364,Z 367.337,A -85,B 0,C 180,E1 -10374.489,E2 -10374.489} C_VEL
LIN {X 0,Y 413.021,Z 355.565,A -85,B 0,C 180,E1 -10377.075,E2 -10377.075} C_VEL
LIN {X 0,Y 411.287,Z 348.049,A -85,B 0,C 180,E1 -10378.826,E2 -10378.826} C_VEL
LIN {X 0,Y 411.169,Z 347.891,A -85,B 0,C 180,E1 -10381.995,E2 -10381.995} C_VEL
LIN {X 0,Y 411.195,Z 347.882,A -85,B 0,C 180,E1 -10385.527,E2 -10385.527} C_VEL
LIN {X 0,Y 411.227,Z 347.878,A -85,B 0,C 180,E1 -10389.221,E2 -10389.221} C_VEL
LIN {X 0,Y 411.227,Z 347.884,A -85,B 0,C 180,E1 -10392.702,E2 -10392.702} C_VEL
LIN {X 0,Y 411.233,Z 347.867,A -85,B 0,C 180,E1 -10395.869,E2 -10395.869} C_VEL
LIN {X 0,Y 411.203,Z 347.887,A -85,B 0,C 180,E1 -10398.763,E2 -10398.763} C_VEL
LIN {X 0,Y 411.197,Z 347.862,A -85,B 0,C 180,E1 -10402.026,E2 -10402.026} C_VEL
LIN {X 0,Y 411.198,Z 347.89,A -85,B 0,C 180,E1 -10405.666,E2 -10405.666} C_VEL
LIN {X 0,Y 411.189,Z 347.872,A -85,B 0,C 180,E1 -10409.152,E2 -10409.152} C_VEL
LIN {X 0,Y 411.25,Z 347.861,A -85,B 0,C 180,E1 -10412.522,E2 -10412.522} C_VEL
LIN {X 0,Y 411.219,Z 347.888,A -85,B 0,C 180,E1 -10415.784,E2 -10415.784} C_VEL
LIN {X 0,Y 411.188,Z 347.88,A -85,B 0,C 180,E1 -10418.965,E2 -10418.965} C_VEL
LIN {X 0,Y 411.242,Z 347.88,A -85,B 0,C 180,E1 -10422.084,E2 -10422.084} C_VEL
LIN {X 0,Y 411.252,Z 347.871,A -85,B 0,C 180,E1 -10425.147,E2 -10425.147} C_VEL
LIN {X 0,Y 411.29,Z 347.872,A -85,B 0,C 180,E1 -10428.167,E2 -10428.167} C_VEL
LIN {X 0,Y 411.471,Z 347.848,A -85,B 0,C 180,E1 -10432.146,E2 -10432.146} C_VEL
LIN {X 0,Y 411.467,Z 347.852,A -85,B 0,C 180,E1 -10434.118,E2 -10434.118} C_VEL
LIN {X 0,Y 411.504,Z 347.843,A -85,B 0,C 180,E1 -10438.042,E2 -10438.042} C_VEL
LIN {X 0,Y 411.635,Z 347.832,A -85,B 0,C 180,E1 -10440,E2 -10440} C_VEL
LIN {X 0,Y 411.458,Z 347.846,A -85,B 0,C 180,E1 -10442.937,E2 -10442.937} C_VEL
LIN {X 0,Y 411.451,Z 347.859,A -85,B 0,C 180,E1 -10446.867,E2 -10446.867} C_VEL
LIN {X 0,Y 411.299,Z 347.86,A -85,B 0,C 180,E1 -10449.839,E2 -10449.839} C_VEL
LIN {X 0,Y 411.302,Z 347.872,A -85,B 0,C 180,E1 -10453.11,E2 -10453.11} C_VEL
LIN {X 0,Y 411.246,Z 347.877,A -85,B 0,C 180,E1 -10456.889,E2 -10456.889} C_VEL
LIN {X 0,Y 411.22,Z 347.881,A -85,B 0,C 180,E1 -10459.987,E2 -10459.987} C_VEL
LIN {X 0,Y 411.194,Z 347.888,A -85,B 0,C 180,E1 -10463.148,E2 -10463.148} C_VEL
LIN {X 0,Y 411.229,Z 347.873,A -85,B 0,C 180,E1 -10466.381,E2 -10466.381} C_VEL
LIN {X 0,Y 411.19,Z 347.856,A -85,B 0,C 180,E1 -10469.713,E2 -10469.713} C_VEL
LIN {X 0,Y 411.197,Z 347.888,A -85,B 0,C 180,E1 -10473.157,E2 -10473.157} C_VEL
LIN {X 0,Y 411.187,Z 347.87,A -85,B 0,C 180,E1 -10476.554,E2 -10476.554} C_VEL
LIN {X 0,Y 411.22,Z 347.875,A -85,B 0,C 180,E1 -10479.731,E2 -10479.731} C_VEL
LIN {X 0,Y 411.223,Z 347.879,A -85,B 0,C 180,E1 -10483.127,E2 -10483.127} C_VEL
LIN {X 0,Y 411.232,Z 347.871,A -85,B 0,C 180,E1 -10485.872,E2 -10485.872} C_VEL
LIN {X 0,Y 411.203,Z 347.883,A -85,B 0,C 180,E1 -10488.765,E2 -10488.765} C_VEL
LIN {X 0,Y 411.199,Z 347.891,A -85,B 0,C 180,E1 -10492.029,E2 -10492.029} C_VEL
LIN {X 0,Y 411.202,Z 347.89,A -85,B 0,C 180,E1 -10495.668,E2 -10495.668} C_VEL
LIN {X 0,Y 411.197,Z 347.885,A -85,B 0,C 180,E1 -10499.155,E2 -10499.155} C_VEL
LIN {X 0,Y 411.264,Z 347.956,A -85,B 0,C 180,E1 -10501.172,E2 -10501.172} C_VEL
LIN {X 0,Y 413.249,Z 356.658,A -85,B 0,C 180,E1 -10503.214,E2 -10503.214} C_VEL
LIN {X 0,Y 415.327,Z 367.117,A -85,B 0,C 180,E1 -10505.509,E2 -10505.509} C_VEL
LIN {X 0,Y 415.03,Z 372.287,A -85,B 0,C 180,E1 -10506.49,E2 -10506.49} C_VEL
LIN {X 0,Y 419.717,Z 395.163,A -85,B 0,C 180,E1 -10507.212,E2 -10507.212} C_VEL
LIN {X 0,Y 420.532,Z 400.544,A -85,B 0,C 180,E1 -10507.357,E2 -10507.357} C_VEL
LIN {X 0,Y 419.174,Z 492.156,A -85,B 0,C 180,E1 -10508.936,E2 -10508.936} C_VEL
LIN {X 0,Y 418.728,Z 512.333,A -85,B 0,C 180,E1 -10509.331,E2 -10509.331} C_VEL
LIN {X 0,Y 418.128,Z 526.768,A -85,B 0,C 180,E1 -10509.814,E2 -10509.814} C_VEL
LIN {X 0,Y 417.413,Z 540.311,A -85,B 0,C 180,E1 -10510.467,E2 -10510.467} C_VEL
LIN {X 0,Y 416.479,Z 553.469,A -85,B 0,C 180,E1 -10511.301,E2 -10511.301} C_VEL
LIN {X 0,Y 415.492,Z 565.574,A -85,B 0,C 180,E1 -10512.275,E2 -10512.275} C_VEL
LIN {X 0,Y 414.366,Z 577.782,A -85,B 0,C 180,E1 -10513.497,E2 -10513.497} C_VEL
LIN {X 0,Y 413.39,Z 587.861,A -85,B 0,C 180,E1 -10514.723,E2 -10514.723} C_VEL
LIN {X 0,Y 412.412,Z 597.877,A -85,B 0,C 180,E1 -10516.199,E2 -10516.199} C_VEL
LIN {X 0,Y 411.759,Z 606.194,A -85,B 0,C 180,E1 -10517.682,E2 -10517.682} C_VEL
LIN {X 0,Y 410.983,Z 614.143,A -85,B 0,C 180,E1 -10519.408,E2 -10519.408} C_VEL
LIN {X 0,Y 410.498,Z 620.539,A -85,B 0,C 180,E1 -10521.138,E2 -10521.138} C_VEL
LIN {X 0,Y 410.172,Z 626.211,A -85,B 0,C 180,E1 -10523.113,E2 -10523.113} C_VEL
LIN {X 0,Y 410.028,Z 630.326,A -85,B 0,C 180,E1 -10525.085,E2 -10525.085} C_VEL
LIN {X 0,Y 409.888,Z 633.009,A -85,B 0,C 180,E1 -10527.053,E2 -10527.053} C_VEL
LIN {X 0,Y 409.916,Z 634.336,A -85,B 0,C 180,E1 -10529.019,E2 -10529.019} C_VEL
LIN {X 0,Y 409.916,Z 634.332,A -85,B 0,C 180,E1 -10530.984,E2 -10530.984} C_VEL
LIN {X 0,Y 409.888,Z 632.998,A -85,B 0,C 180,E1 -10532.95,E2 -10532.95} C_VEL
LIN {X 0,Y 410.026,Z 630.309,A -85,B 0,C 180,E1 -10534.918,E2 -10534.918} C_VEL
LIN {X 0,Y 410.163,Z 626.191,A -85,B 0,C 180,E1 -10536.89,E2 -10536.89} C_VEL
LIN {X 0,Y 410.501,Z 620.515,A -85,B 0,C 180,E1 -10538.865,E2 -10538.865} C_VEL
LIN {X 0,Y 410.984,Z 614.11,A -85,B 0,C 180,E1 -10540.594,E2 -10540.594} C_VEL
LIN {X 0,Y 411.746,Z 606.154,A -85,B 0,C 180,E1 -10542.32,E2 -10542.32} C_VEL
LIN {X 0,Y 412.457,Z 597.828,A -85,B 0,C 180,E1 -10543.802,E2 -10543.802} C_VEL
LIN {X 0,Y 413.381,Z 587.8,A -85,B 0,C 180,E1 -10545.28,E2 -10545.28} C_VEL
LIN {X 0,Y 414.443,Z 576.612,A -85,B 0,C 180,E1 -10546.629,E2 -10546.629} C_VEL
LIN {X 0,Y 415.605,Z 564.048,A -85,B 0,C 180,E1 -10547.849,E2 -10547.849} C_VEL
LIN {X 0,Y 416.57,Z 551.639,A -85,B 0,C 180,E1 -10548.82,E2 -10548.82} C_VEL
LIN {X 0,Y 417.534,Z 537.625,A -85,B 0,C 180,E1 -10549.674,E2 -10549.674} C_VEL
LIN {X 0,Y 418.221,Z 524.272,A -85,B 0,C 180,E1 -10550.28,E2 -10550.28} C_VEL
LIN {X 0,Y 418.809,Z 509.723,A -85,B 0,C 180,E1 -10550.732,E2 -10550.732} C_VEL
LIN {X 0,Y 420.474,Z 405.769,A -85,B 0,C 180,E1 -10552.545,E2 -10552.545} C_VEL
LIN {X 0,Y 420.418,Z 399.096,A -85,B 0,C 180,E1 -10552.669,E2 -10552.669} C_VEL
LIN {X 0,Y 415.216,Z 373.218,A -85,B 0,C 180,E1 -10553.456,E2 -10553.456} C_VEL
LIN {X 0,Y 415.081,Z 371.742,A -85,B 0,C 180,E1 -10553.58,E2 -10553.58} C_VEL
LIN {X 0,Y 415.313,Z 367.062,A -85,B 0,C 180,E1 -10554.495,E2 -10554.495} C_VEL
LIN {X 0,Y 412.943,Z 355.29,A -85,B 0,C 180,E1 -10557.083,E2 -10557.083} C_VEL
LIN {X 0,Y 411.289,Z 348.029,A -85,B 0,C 180,E1 -10558.767,E2 -10558.767} C_VEL
LIN {X 0,Y 411.17,Z 347.894,A -85,B 0,C 180,E1 -10561.998,E2 -10561.998} C_VEL
LIN {X 0,Y 411.216,Z 347.888,A -85,B 0,C 180,E1 -10564.879,E2 -10564.879} C_VEL
LIN {X 0,Y 411.214,Z 347.888,A -85,B 0,C 180,E1 -10568.17,E2 -10568.17} C_VEL
LIN {X 0,Y 411.168,Z 347.891,A -85,B 0,C 180,E1 -10571.229,E2 -10571.229} C_VEL
LIN {X 0,Y 411.18,Z 347.89,A -85,B 0,C 180,E1 -10574.491,E2 -10574.491} C_VEL
LIN {X 0,Y 411.182,Z 347.892,A -85,B 0,C 180,E1 -10578.195,E2 -10578.195} C_VEL
LIN {X 0,Y 411.222,Z 347.886,A -85,B 0,C 180,E1 -10580.776,E2 -10580.776} C_VEL
LIN {X 0,Y 411.203,Z 347.89,A -85,B 0,C 180,E1 -10584.472,E2 -10584.472} C_VEL
LIN {X 0,Y 411.246,Z 348.1,A -85,B 0,C 180,E1 -10587.612,E2 -10587.612} C_VEL
LIN {X 0,Y 414.632,Z 358.464,A -85,B 0,C 180,E1 -10589.821,E2 -10589.821} C_VEL
LIN {X 0,Y 417.007,Z 367.948,A -85,B 0,C 180,E1 -10591.646,E2 -10591.646} C_VEL
LIN {X 0,Y 417.818,Z 372.345,A -85,B 0,C 180,E1 -10592.447,E2 -10592.447} C_VEL
LIN {X 0,Y 416.925,Z 387.426,A -85,B 0,C 180,E1 -10594.809,E2 -10594.809} C_VEL
LIN {X 0,Y 415.704,Z 407.503,A -85,B 0,C 180,E1 -10597.904,E2 -10597.904} C_VEL
LIN {X 0,Y 415.039,Z 420.575,A -85,B 0,C 180,E1 -10599.882,E2 -10599.882} C_VEL
LIN {X 0,Y 417.687,Z 435.436,A -85,B 0,C 180,E1 -10600.481,E2 -10600.481} C_VEL
LIN {X 0,Y 418.589,Z 443.869,A -85,B 0,C 180,E1 -10600.764,E2 -10600.764} C_VEL
LIN {X 0,Y 416.396,Z 521.732,A -85,B 0,C 180,E1 -10602.567,E2 -10602.567} C_VEL
LIN {X 0,Y 415.92,Z 537.197,A -85,B 0,C 180,E1 -10602.99,E2 -10602.99} C_VEL
LIN {X 0,Y 415.335,Z 550.025,A -85,B 0,C 180,E1 -10603.535,E2 -10603.535} C_VEL
LIN {X 0,Y 414.617,Z 562.461,A -85,B 0,C 180,E1 -10604.264,E2 -10604.264} C_VEL
LIN {X 0,Y 413.881,Z 573.788,A -85,B 0,C 180,E1 -10605.118,E2 -10605.118} C_VEL
LIN {X 0,Y 413.038,Z 585.32,A -85,B 0,C 180,E1 -10606.219,E2 -10606.219} C_VEL
LIN {X 0,Y 412.271,Z 595.668,A -85,B 0,C 180,E1 -10607.447,E2 -10607.447} C_VEL
LIN {X 0,Y 411.613,Z 604.089,A -85,B 0,C 180,E1 -10608.676,E2 -10608.676} C_VEL
LIN {X 0,Y 411.038,Z 612.329,A -85,B 0,C 180,E1 -10610.155,E2 -10610.155} C_VEL
LIN {X 0,Y 410.573,Z 618.974,A -85,B 0,C 180,E1 -10611.634,E2 -10611.634} C_VEL
LIN {X 0,Y 410.255,Z 624.236,A -85,B 0,C 180,E1 -10613.113,E2 -10613.113} C_VEL
LIN {X 0,Y 410.138,Z 628.284,A -85,B 0,C 180,E1 -10614.592,E2 -10614.592} C_VEL
LIN {X 0,Y 409.944,Z 631.243,A -85,B 0,C 180,E1 -10616.068,E2 -10616.068} C_VEL
LIN {X 0,Y 409.911,Z 632.629,A -85,B 0,C 180,E1 -10617.052,E2 -10617.052} C_VEL
LIN {X 0,Y 409.946,Z 633.602,A -85,B 0,C 180,E1 -10618.035,E2 -10618.035} C_VEL
LIN {X 0,Y 409.92,Z 634.15,A -85,B 0,C 180,E1 -10619.018,E2 -10619.018} C_VEL
LIN {X 0,Y 409.889,Z 634.23,A -85,B 0,C 180,E1 -10620,E2 -10620} C_VEL
LIN {X 0,Y 409.92,Z 633.897,A -85,B 0,C 180,E1 -10620.982,E2 -10620.982} C_VEL
LIN {X 0,Y 409.929,Z 633.15,A -85,B 0,C 180,E1 -10621.965,E2 -10621.965} C_VEL
LIN {X 0,Y 409.894,Z 631.924,A -85,B 0,C 180,E1 -10622.949,E2 -10622.949} C_VEL
LIN {X 0,Y 410.003,Z 629.27,A -85,B 0,C 180,E1 -10624.424,E2 -10624.424} C_VEL
LIN {X 0,Y 410.082,Z 625.534,A -85,B 0,C 180,E1 -10625.902,E2 -10625.902} C_VEL
LIN {X 0,Y 410.286,Z 620.62,A -85,B 0,C 180,E1 -10627.381,E2 -10627.381} C_VEL
LIN {X 0,Y 410.567,Z 614.383,A -85,B 0,C 180,E1 -10628.862,E2 -10628.862} C_VEL
LIN {X 0,Y 410.964,Z 606.561,A -85,B 0,C 180,E1 -10630.344,E2 -10630.344} C_VEL
LIN {X 0,Y 411.553,Z 596.764,A -85,B 0,C 180,E1 -10631.825,E2 -10631.825} C_VEL
LIN {X 0,Y 412.194,Z 586.64,A -85,B 0,C 180,E1 -10633.051,E2 -10633.051} C_VEL
LIN {X 0,Y 412.816,Z 575.203,A -85,B 0,C 180,E1 -10634.165,E2 -10634.165} C_VEL
LIN {X 0,Y 413.349,Z 564.049,A -85,B 0,C 180,E1 -10635.028,E2 -10635.028} C_VEL
LIN {X 0,Y 414.04,Z 550.549,A -85,B 0,C 180,E1 -10635.822,E2 -10635.822} C_VEL
LIN {X 0,Y 414.475,Z 537.456,A -85,B 0,C 180,E1 -10636.374,E2 -10636.374} C_VEL
LIN {X 0,Y 414.821,Z 523.882,A -85,B 0,C 180,E1 -10636.739,E2 -10636.739} C_VEL
LIN {X 0,Y 416.208,Z 441.988,A -85,B 0,C 180,E1 -10638.448,E2 -10638.448} C_VEL
LIN {X 0,Y 413.39,Z 420.689,A -85,B 0,C 180,E1 -10639.039,E2 -10639.039} C_VEL
LIN {X 0,Y 414.316,Z 400.078,A -85,B 0,C 180,E1 -10642.174,E2 -10642.174} C_VEL
LIN {X 0,Y 415.355,Z 379.802,A -85,B 0,C 180,E1 -10645.293,E2 -10645.293} C_VEL
LIN {X 0,Y 415.83,Z 369.432,A -85,B 0,C 180,E1 -10646.893,E2 -10646.893} C_VEL
LIN {X 0,Y 414.153,Z 360.609,A -85,B 0,C 180,E1 -10648.369,E2 -10648.369} C_VEL
LIN {X 0,Y 411.241,Z 348.01,A -85,B 0,C 180,E1 -10650.576,E2 -10650.576} C_VEL
LIN {X 0,Y 411.211,Z 347.89,A -85,B 0,C 180,E1 -10654.333,E2 -10654.333} C_VEL
LIN {X 0,Y 411.197,Z 347.891,A -85,B 0,C 180,E1 -10657.974,E2 -10657.974} C_VEL
LIN {X 0,Y 411.169,Z 347.891,A -85,B 0,C 180,E1 -10661.228,E2 -10661.228} C_VEL
LIN {X 0,Y 411.181,Z 347.872,A -85,B 0,C 180,E1 -10664.49,E2 -10664.49} C_VEL
LIN {X 0,Y 411.183,Z 347.893,A -85,B 0,C 180,E1 -10668.194,E2 -10668.194} C_VEL
LIN {X 0,Y 411.226,Z 347.876,A -85,B 0,C 180,E1 -10670.776,E2 -10670.776} C_VEL
LIN {X 0,Y 411.205,Z 347.881,A -85,B 0,C 180,E1 -10674.471,E2 -10674.471} C_VEL
LIN {X 0,Y 411.213,Z 347.882,A -85,B 0,C 180,E1 -10676.873,E2 -10676.873} C_VEL
LIN {X 0,Y 411.238,Z 347.858,A -85,B 0,C 180,E1 -10680.643,E2 -10680.643} C_VEL
LIN {X 0,Y 411.317,Z 348.093,A -85,B 0,C 180,E1 -10681.296,E2 -10681.296} C_VEL
LIN {X 0,Y 414.052,Z 360.427,A -85,B 0,C 180,E1 -10684.107,E2 -10684.107} C_VEL
LIN {X 0,Y 415.38,Z 368.148,A -85,B 0,C 180,E1 -10685.775,E2 -10685.775} C_VEL
LIN {X 0,Y 415.051,Z 372.357,A -85,B 0,C 180,E1 -10686.55,E2 -10686.55} C_VEL
LIN {X 0,Y 420.041,Z 397.029,A -85,B 0,C 180,E1 -10687.317,E2 -10687.317} C_VEL
LIN {X 0,Y 420.506,Z 401.688,A -85,B 0,C 180,E1 -10687.428,E2 -10687.428} C_VEL
LIN {X 0,Y 419.155,Z 493.521,A -85,B 0,C 180,E1 -10689.012,E2 -10689.012} C_VEL
LIN {X 0,Y 418.399,Z 499.375,A -85,B 0,C 180,E1 -10689.077,E2 -10689.077} C_VEL
LIN {X 0,Y 415.418,Z 508.861,A -85,B 0,C 180,E1 -10689.114,E2 -10689.114} C_VEL
LIN {X 0,Y 412.406,Z 518.25,A -85,B 0,C 180,E1 -10689.231,E2 -10689.231} C_VEL
LIN {X 0,Y 411.564,Z 523.94,A -85,B 0,C 180,E1 -10689.408,E2 -10689.408} C_VEL
LIN {X 0,Y 410.873,Z 536.84,A -85,B 0,C 180,E1 -10689.994,E2 -10689.994} C_VEL
LIN {X 0,Y 410.058,Z 549.422,A -85,B 0,C 180,E1 -10690.751,E2 -10690.751} C_VEL
LIN {X 0,Y 409.025,Z 562.123,A -85,B 0,C 180,E1 -10691.724,E2 -10691.724} C_VEL
LIN {X 0,Y 407.748,Z 575.027,A -85,B 0,C 180,E1 -10692.96,E2 -10692.96} C_VEL
LIN {X 0,Y 406.739,Z 585.559,A -85,B 0,C 180,E1 -10694.207,E2 -10694.207} C_VEL
LIN {X 0,Y 405.659,Z 596.018,A -85,B 0,C 180,E1 -10695.706,E2 -10695.706} C_VEL
LIN {X 0,Y 404.931,Z 604.647,A -85,B 0,C 180,E1 -10697.214,E2 -10697.214} C_VEL
LIN {X 0,Y 404.054,Z 612.919,A -85,B 0,C 180,E1 -10698.968,E2 -10698.968} C_VEL
LIN {X 0,Y 403.605,Z 618.687,A -85,B 0,C 180,E1 -10700.477,E2 -10700.477} C_VEL
LIN {X 0,Y 403.221,Z 623.43,A -85,B 0,C 180,E1 -10701.984,E2 -10701.984} C_VEL
LIN {X 0,Y 402.988,Z 628.339,A -85,B 0,C 180,E1 -10703.992,E2 -10703.992} C_VEL
LIN {X 0,Y 402.849,Z 631.76,A -85,B 0,C 180,E1 -10705.997,E2 -10705.997} C_VEL
LIN {X 0,Y 402.824,Z 633.796,A -85,B 0,C 180,E1 -10707.999,E2 -10707.999} C_VEL
LIN {X 0,Y 402.814,Z 634.498,A -85,B 0,C 180,E1 -10709.999,E2 -10709.999} C_VEL
LIN {X 0,Y 402.822,Z 633.872,A -85,B 0,C 180,E1 -10711.998,E2 -10711.998} C_VEL
LIN {X 0,Y 402.848,Z 631.907,A -85,B 0,C 180,E1 -10714,E2 -10714} C_VEL
LIN {X 0,Y 402.986,Z 628.551,A -85,B 0,C 180,E1 -10716.005,E2 -10716.005} C_VEL
LIN {X 0,Y 403.216,Z 623.706,A -85,B 0,C 180,E1 -10718.014,E2 -10718.014} C_VEL
LIN {X 0,Y 403.752,Z 617.23,A -85,B 0,C 180,E1 -10720.023,E2 -10720.023} C_VEL
LIN {X 0,Y 404.408,Z 610.02,A -85,B 0,C 180,E1 -10721.781,E2 -10721.781} C_VEL
LIN {X 0,Y 405.084,Z 602.244,A -85,B 0,C 180,E1 -10723.33,E2 -10723.33} C_VEL
LIN {X 0,Y 405.962,Z 593.395,A -85,B 0,C 180,E1 -10724.793,E2 -10724.793} C_VEL
LIN {X 0,Y 407.033,Z 582.409,A -85,B 0,C 180,E1 -10726.293,E2 -10726.293} C_VEL
LIN {X 0,Y 408.184,Z 571.214,A -85,B 0,C 180,E1 -10727.535,E2 -10727.535} C_VEL
LIN {X 0,Y 409.265,Z 558.829,A -85,B 0,C 180,E1 -10728.651,E2 -10728.651} C_VEL
LIN {X 0,Y 410.268,Z 546.761,A -85,B 0,C 180,E1 -10729.522,E2 -10729.522} C_VEL
LIN {X 0,Y 411.054,Z 533.841,A -85,B 0,C 180,E1 -10730.255,E2 -10730.255} C_VEL
LIN {X 0,Y 411.821,Z 519.769,A -85,B 0,C 180,E1 -10730.836,E2 -10730.836} C_VEL
LIN {X 0,Y 412.346,Z 504.929,A -85,B 0,C 180,E1 -10731.233,E2 -10731.233} C_VEL
LIN {X 0,Y 413.966,Z 400.373,A -85,B 0,C 180,E1 -10733.071,E2 -10733.071} C_VEL
LIN {X 0,Y 408.595,Z 374.114,A -85,B 0,C 180,E1 -10733.886,E2 -10733.886} C_VEL
LIN {X 0,Y 408.264,Z 372.036,A -85,B 0,C 180,E1 -10733.996,E2 -10733.996} C_VEL
LIN {X 0,Y 408.445,Z 368.643,A -85,B 0,C 180,E1 -10734.66,E2 -10734.66} C_VEL
LIN {X 0,Y 406.089,Z 356.871,A -85,B 0,C 180,E1 -10737.297,E2 -10737.297} C_VEL
LIN {X 0,Y 404.258,Z 349.092,A -85,B 0,C 180,E1 -10739.127,E2 -10739.127} C_VEL
LIN {X 0,Y 404.207,Z 348.744,A -85,B 0,C 180,E1 -10739.367,E2 -10739.367} C_VEL
LIN {X 0,Y 404.14,Z 348.761,A -85,B 0,C 180,E1 -10742.62,E2 -10742.62} C_VEL
LIN {X 0,Y 404.178,Z 348.759,A -85,B 0,C 180,E1 -10745.189,E2 -10745.189} C_VEL
LIN {X 0,Y 404.159,Z 348.761,A -85,B 0,C 180,E1 -10748.754,E2 -10748.754} C_VEL
LIN {X 0,Y 404.186,Z 348.759,A -85,B 0,C 180,E1 -10751.609,E2 -10751.609} C_VEL
LIN {X 0,Y 404.194,Z 348.744,A -85,B 0,C 180,E1 -10754.529,E2 -10754.529} C_VEL
LIN {X 0,Y 404.204,Z 348.754,A -85,B 0,C 180,E1 -10757.304,E2 -10757.304} C_VEL
LIN {X 0,Y 404.161,Z 348.757,A -85,B 0,C 180,E1 -10759.954,E2 -10759.954} C_VEL
LIN {X 0,Y 404.133,Z 348.745,A -85,B 0,C 180,E1 -10763.123,E2 -10763.123} C_VEL
LIN {X 0,Y 404.136,Z 348.769,A -85,B 0,C 180,E1 -10766.187,E2 -10766.187} C_VEL
LIN {X 0,Y 404.144,Z 348.738,A -85,B 0,C 180,E1 -10769.715,E2 -10769.715} C_VEL
LIN {X 0,Y 404.186,Z 348.743,A -85,B 0,C 180,E1 -10773.122,E2 -10773.122} C_VEL
LIN {X 0,Y 404.168,Z 348.764,A -85,B 0,C 180,E1 -10775.334,E2 -10775.334} C_VEL
LIN {X 0,Y 404.13,Z 348.758,A -85,B 0,C 180,E1 -10778.58,E2 -10778.58} C_VEL
LIN {X 0,Y 404.2,Z 348.759,A -85,B 0,C 180,E1 -10781.761,E2 -10781.761} C_VEL
LIN {X 0,Y 404.198,Z 348.747,A -85,B 0,C 180,E1 -10784.882,E2 -10784.882} C_VEL
LIN {X 0,Y 404.261,Z 348.749,A -85,B 0,C 180,E1 -10787.959,E2 -10787.959} C_VEL
LIN {X 0,Y 404.422,Z 348.726,A -85,B 0,C 180,E1 -10792.099,E2 -10792.099} C_VEL
LIN {X 0,Y 404.415,Z 348.73,A -85,B 0,C 180,E1 -10794.015,E2 -10794.015} C_VEL
LIN {X 0,Y 404.473,Z 348.719,A -85,B 0,C 180,E1 -10798.008,E2 -10798.008} C_VEL
LIN {X 0,Y 404.605,Z 348.708,A -85,B 0,C 180,E1 -10800,E2 -10800} C_VEL
LIN {X 0,Y 404.415,Z 348.722,A -85,B 0,C 180,E1 -10802.988,E2 -10802.988} C_VEL
LIN {X 0,Y 404.401,Z 348.735,A -85,B 0,C 180,E1 -10806.987,E2 -10806.987} C_VEL
LIN {X 0,Y 404.261,Z 348.737,A -85,B 0,C 180,E1 -10810.012,E2 -10810.012} C_VEL
LIN {X 0,Y 404.255,Z 348.749,A -85,B 0,C 180,E1 -10813.212,E2 -10813.212} C_VEL
LIN {X 0,Y 404.205,Z 348.756,A -85,B 0,C 180,E1 -10817.007,E2 -10817.007} C_VEL
LIN {X 0,Y 404.177,Z 348.757,A -85,B 0,C 180,E1 -10820.351,E2 -10820.351} C_VEL
LIN {X 0,Y 404.16,Z 348.763,A -85,B 0,C 180,E1 -10823.575,E2 -10823.575} C_VEL
LIN {X 0,Y 404.174,Z 348.758,A -85,B 0,C 180,E1 -10825.767,E2 -10825.767} C_VEL
LIN {X 0,Y 404.185,Z 348.731,A -85,B 0,C 180,E1 -10828,E2 -10828} C_VEL
LIN {X 0,Y 404.13,Z 348.758,A -85,B 0,C 180,E1 -10831.559,E2 -10831.559} C_VEL
LIN {X 0,Y 404.176,Z 348.758,A -85,B 0,C 180,E1 -10835.017,E2 -10835.017} C_VEL
LIN {X 0,Y 404.155,Z 348.744,A -85,B 0,C 180,E1 -10838.757,E2 -10838.757} C_VEL
LIN {X 0,Y 404.184,Z 348.762,A -85,B 0,C 180,E1 -10841.612,E2 -10841.612} C_VEL
LIN {X 0,Y 404.193,Z 348.741,A -85,B 0,C 180,E1 -10844.531,E2 -10844.531} C_VEL
LIN {X 0,Y 404.204,Z 348.759,A -85,B 0,C 180,E1 -10847.307,E2 -10847.307} C_VEL
LIN {X 0,Y 404.162,Z 348.753,A -85,B 0,C 180,E1 -10849.957,E2 -10849.957} C_VEL
LIN {X 0,Y 404.135,Z 348.767,A -85,B 0,C 180,E1 -10853.125,E2 -10853.125} C_VEL
LIN {X 0,Y 404.14,Z 348.767,A -85,B 0,C 180,E1 -10856.189,E2 -10856.189} C_VEL
LIN {X 0,Y 404.151,Z 348.749,A -85,B 0,C 180,E1 -10859.717,E2 -10859.717} C_VEL
LIN {X 0,Y 404.234,Z 348.953,A -85,B 0,C 180,E1 -10860.871,E2 -10860.871} C_VEL
LIN {X 0,Y 406.599,Z 359.274,A -85,B 0,C 180,E1 -10863.296,E2 -10863.296} C_VEL
LIN {X 0,Y 408.422,Z 368.426,A -85,B 0,C 180,E1 -10865.338,E2 -10865.338} C_VEL
LIN {X 0,Y 408.291,Z 372.395,A -85,B 0,C 180,E1 -10866.084,E2 -10866.084} C_VEL
LIN {X 0,Y 413.466,Z 397.758,A -85,B 0,C 180,E1 -10866.896,E2 -10866.896} C_VEL
LIN {X 0,Y 413.994,Z 400.789,A -85,B 0,C 180,E1 -10866.983,E2 -10866.983} C_VEL
LIN {X 0,Y 412.261,Z 508.861,A -85,B 0,C 180,E1 -10868.894,E2 -10868.894} C_VEL
LIN {X 0,Y 411.666,Z 522.969,A -85,B 0,C 180,E1 -10869.32,E2 -10869.32} C_VEL
LIN {X 0,Y 410.922,Z 536.654,A -85,B 0,C 180,E1 -10869.934,E2 -10869.934} C_VEL
LIN {X 0,Y 410.005,Z 550.366,A -85,B 0,C 180,E1 -10870.766,E2 -10870.766} C_VEL
LIN {X 0,Y 409.003,Z 562.73,A -85,B 0,C 180,E1 -10871.726,E2 -10871.726} C_VEL
LIN {X 0,Y 407.832,Z 574.35,A -85,B 0,C 180,E1 -10872.837,E2 -10872.837} C_VEL
LIN {X 0,Y 406.895,Z 584.021,A -85,B 0,C 180,E1 -10873.959,E2 -10873.959} C_VEL
LIN {X 0,Y 405.785,Z 594.737,A -85,B 0,C 180,E1 -10875.457,E2 -10875.457} C_VEL
LIN {X 0,Y 405.018,Z 603.58,A -85,B 0,C 180,E1 -10876.964,E2 -10876.964} C_VEL
LIN {X 0,Y 404.156,Z 612.054,A -85,B 0,C 180,E1 -10878.72,E2 -10878.72} C_VEL
LIN {X 0,Y 403.587,Z 618.877,A -85,B 0,C 180,E1 -10880.479,E2 -10880.479} C_VEL
LIN {X 0,Y 403.215,Z 623.579,A -85,B 0,C 180,E1 -10881.986,E2 -10881.986} C_VEL
LIN {X 0,Y 403.005,Z 628.455,A -85,B 0,C 180,E1 -10883.995,E2 -10883.995} C_VEL
LIN {X 0,Y 402.848,Z 631.841,A -85,B 0,C 180,E1 -10886,E2 -10886} C_VEL
LIN {X 0,Y 402.822,Z 633.84,A -85,B 0,C 180,E1 -10888.002,E2 -10888.002} C_VEL
LIN {X 0,Y 402.813,Z 634.5,A -85,B 0,C 180,E1 -10890.001,E2 -10890.001} C_VEL
LIN {X 0,Y 402.822,Z 633.832,A -85,B 0,C 180,E1 -10892.001,E2 -10892.001} C_VEL
LIN {X 0,Y 402.848,Z 631.825,A -85,B 0,C 180,E1 -10894.003,E2 -10894.003} C_VEL
LIN {X 0,Y 402.987,Z 628.434,A -85,B 0,C 180,E1 -10896.008,E2 -10896.008} C_VEL
LIN {X 0,Y 403.217,Z 623.557,A -85,B 0,C 180,E1 -10898.017,E2 -10898.017} C_VEL
LIN {X 0,Y 403.759,Z 617.039,A -85,B 0,C 180,E1 -10900.025,E2 -10900.025} C_VEL
LIN {X 0,Y 404.426,Z 609.783,A -85,B 0,C 180,E1 -10901.783,E2 -10901.783} C_VEL
LIN {X 0,Y 405.111,Z 601.944,A -85,B 0,C 180,E1 -10903.334,E2 -10903.334} C_VEL
LIN {X 0,Y 405.959,Z 593.05,A -85,B 0,C 180,E1 -10904.796,E2 -10904.796} C_VEL
LIN {X 0,Y 407.044,Z 581.979,A -85,B 0,C 180,E1 -10906.295,E2 -10906.295} C_VEL
LIN {X 0,Y 408.225,Z 570.669,A -85,B 0,C 180,E1 -10907.536,E2 -10907.536} C_VEL
LIN {X 0,Y 409.322,Z 558.156,A -85,B 0,C 180,E1 -10908.651,E2 -10908.651} C_VEL
LIN {X 0,Y 410.323,Z 545.01,A -85,B 0,C 180,E1 -10909.582,E2 -10909.582} C_VEL
LIN {X 0,Y 411.158,Z 531.454,A -85,B 0,C 180,E1 -10910.318,E2 -10910.318} C_VEL
LIN {X 0,Y 411.888,Z 517.315,A -85,B 0,C 180,E1 -10910.867,E2 -10910.867} C_VEL
LIN {X 0,Y 412.348,Z 502.341,A -85,B 0,C 180,E1 -10911.235,E2 -10911.235} C_VEL
LIN {X 0,Y 413.923,Z 403.957,A -85,B 0,C 180,E1 -10912.955,E2 -10912.955} C_VEL
LIN {X 0,Y 413.76,Z 399.503,A -85,B 0,C 180,E1 -10913.047,E2 -10913.047} C_VEL
LIN {X 0,Y 408.376,Z 372.777,A -85,B 0,C 180,E1 -10913.886,E2 -10913.886} C_VEL
LIN {X 0,Y 408.308,Z 371.74,A -85,B 0,C 180,E1 -10913.996,E2 -10913.996} C_VEL
LIN {X 0,Y 408.402,Z 368.368,A -85,B 0,C 180,E1 -10914.666,E2 -10914.666} C_VEL
LIN {X 0,Y 406.008,Z 356.596,A -85,B 0,C 180,E1 -10917.305,E2 -10917.305} C_VEL
LIN {X 0,Y 404.213,Z 348.833,A -85,B 0,C 180,E1 -10919.163,E2 -10919.163} C_VEL
LIN {X 0,Y 404.146,Z 348.768,A -85,B 0,C 180,E1 -10922.622,E2 -10922.622} C_VEL
LIN {X 0,Y 404.187,Z 348.764,A -85,B 0,C 180,E1 -10925.191,E2 -10925.191} C_VEL
LIN {X 0,Y 404.161,Z 348.767,A -85,B 0,C 180,E1 -10928.757,E2 -10928.757} C_VEL
LIN {X 0,Y 404.127,Z 348.769,A -85,B 0,C 180,E1 -10931.6,E2 -10931.6} C_VEL
LIN {X 0,Y 404.15,Z 348.765,A -85,B 0,C 180,E1 -10934.523,E2 -10934.523} C_VEL
LIN {X 0,Y 404.141,Z 348.771,A -85,B 0,C 180,E1 -10937.296,E2 -10937.296} C_VEL
LIN {X 0,Y 404.174,Z 348.766,A -85,B 0,C 180,E1 -10939.956,E2 -10939.956} C_VEL
LIN {X 0,Y 404.141,Z 348.771,A -85,B 0,C 180,E1 -10943.126,E2 -10943.126} C_VEL
LIN {X 0,Y 404.15,Z 348.769,A -85,B 0,C 180,E1 -10946.188,E2 -10946.188} C_VEL
LIN {X 0,Y 404.215,Z 349.079,A -85,B 0,C 180,E1 -10946.851,E2 -10946.851} C_VEL
LIN {X 0,Y 408.104,Z 360.629,A -85,B 0,C 180,E1 -10949.437,E2 -10949.437} C_VEL
LIN {X 0,Y 410.53,Z 370.247,A -85,B 0,C 180,E1 -10951.358,E2 -10951.358} C_VEL
LIN {X 0,Y 411.377,Z 375.005,A -85,B 0,C 180,E1 -10952.255,E2 -10952.255} C_VEL
LIN {X 0,Y 409.994,Z 395.839,A -85,B 0,C 180,E1 -10955.545,E2 -10955.545} C_VEL
LIN {X 0,Y 408.509,Z 418.436,A -85,B 0,C 180,E1 -10959.085,E2 -10959.085} C_VEL
LIN {X 0,Y 408.483,Z 420.649,A -85,B 0,C 180,E1 -10959.38,E2 -10959.38} C_VEL
LIN {X 0,Y 411.052,Z 434.489,A -85,B 0,C 180,E1 -10959.983,E2 -10959.983} C_VEL
LIN {X 0,Y 412.213,Z 444.659,A -85,B 0,C 180,E1 -10960.347,E2 -10960.347} C_VEL
LIN {X 0,Y 410.034,Z 513.366,A -85,B 0,C 180,E1 -10961.998,E2 -10961.998} C_VEL
LIN {X 0,Y 409.451,Z 534.058,A -85,B 0,C 180,E1 -10962.52,E2 -10962.52} C_VEL
LIN {X 0,Y 408.811,Z 547.697,A -85,B 0,C 180,E1 -10963.072,E2 -10963.072} C_VEL
LIN {X 0,Y 408.051,Z 559.795,A -85,B 0,C 180,E1 -10963.747,E2 -10963.747} C_VEL
LIN {X 0,Y 407.189,Z 573.067,A -85,B 0,C 180,E1 -10964.739,E2 -10964.739} C_VEL
LIN {X 0,Y 406.296,Z 583.727,A -85,B 0,C 180,E1 -10965.743,E2 -10965.743} C_VEL
LIN {X 0,Y 405.527,Z 594.205,A -85,B 0,C 180,E1 -10966.98,E2 -10966.98} C_VEL
LIN {X 0,Y 404.793,Z 602.904,A -85,B 0,C 180,E1 -10968.229,E2 -10968.229} C_VEL
LIN {X 0,Y 404.171,Z 611.378,A -85,B 0,C 180,E1 -10969.733,E2 -10969.733} C_VEL
LIN {X 0,Y 403.633,Z 618.187,A -85,B 0,C 180,E1 -10971.237,E2 -10971.237} C_VEL
LIN {X 0,Y 403.195,Z 624.411,A -85,B 0,C 180,E1 -10972.992,E2 -10972.992} C_VEL
LIN {X 0,Y 403.059,Z 628.41,A -85,B 0,C 180,E1 -10974.497,E2 -10974.497} C_VEL
LIN {X 0,Y 402.869,Z 631.326,A -85,B 0,C 180,E1 -10975.999,E2 -10975.999} C_VEL
LIN {X 0,Y 402.811,Z 632.692,A -85,B 0,C 180,E1 -10977,E2 -10977} C_VEL
LIN {X 0,Y 402.844,Z 633.645,A -85,B 0,C 180,E1 -10978.001,E2 -10978.001} C_VEL
LIN {X 0,Y 402.848,Z 634.15,A -85,B 0,C 180,E1 -10979,E2 -10979} C_VEL
LIN {X 0,Y 402.816,Z 634.203,A -85,B 0,C 180,E1 -10980,E2 -10980} C_VEL
LIN {X 0,Y 402.847,Z 633.845,A -85,B 0,C 180,E1 -10981,E2 -10981} C_VEL
LIN {X 0,Y 402.826,Z 633.055,A -85,B 0,C 180,E1 -10982,E2 -10982} C_VEL
LIN {X 0,Y 402.796,Z 631.791,A -85,B 0,C 180,E1 -10983.001,E2 -10983.001} C_VEL
LIN {X 0,Y 402.931,Z 629.077,A -85,B 0,C 180,E1 -10984.502,E2 -10984.502} C_VEL
LIN {X 0,Y 403.061,Z 624.318,A -85,B 0,C 180,E1 -10986.333,E2 -10986.333} C_VEL
LIN {X 0,Y 403.304,Z 618.327,A -85,B 0,C 180,E1 -10988.014,E2 -10988.014} C_VEL
LIN {X 0,Y 403.636,Z 611.492,A -85,B 0,C 180,E1 -10989.521,E2 -10989.521} C_VEL
LIN {X 0,Y 403.997,Z 604.5,A -85,B 0,C 180,E1 -10990.778,E2 -10990.778} C_VEL
LIN {X 0,Y 404.575,Z 596.078,A -85,B 0,C 180,E1 -10992.032,E2 -10992.032} C_VEL
LIN {X 0,Y 405.227,Z 586.026,A -85,B 0,C 180,E1 -10993.25,E2 -10993.25} C_VEL
LIN {X 0,Y 405.79,Z 575.516,A -85,B 0,C 180,E1 -10994.288,E2 -10994.288} C_VEL
LIN {X 0,Y 406.338,Z 564.482,A -85,B 0,C 180,E1 -10995.165,E2 -10995.165} C_VEL
LIN {X 0,Y 407.047,Z 551.131,A -85,B 0,C 180,E1 -10995.972,E2 -10995.972} C_VEL
LIN {X 0,Y 407.478,Z 538.414,A -85,B 0,C 180,E1 -10996.534,E2 -10996.534} C_VEL
LIN {X 0,Y 407.88,Z 524.045,A -85,B 0,C 180,E1 -10996.936,E2 -10996.936} C_VEL
LIN {X 0,Y 409.285,Z 442.282,A -85,B 0,C 180,E1 -10998.687,E2 -10998.687} C_VEL
LIN {X 0,Y 406.434,Z 420.58,A -85,B 0,C 180,E1 -10999.312,E2 -10999.312} C_VEL
LIN {X 0,Y 407.373,Z 401.145,A -85,B 0,C 180,E1 -11002.306,E2 -11002.306} C_VEL
LIN {X 0,Y 408.459,Z 380.703,A -85,B 0,C 180,E1 -11005.477,E2 -11005.477} C_VEL
LIN {X 0,Y 408.9,Z 370.356,A -85,B 0,C 180,E1 -11007.095,E2 -11007.095} C_VEL
LIN {X 0,Y 406.292,Z 357.971,A -85,B 0,C 180,E1 -11009.214,E2 -11009.214} C_VEL
LIN {X 0,Y 404.205,Z 348.887,A -85,B 0,C 180,E1 -11010.841,E2 -11010.841} C_VEL
LIN {X 0,Y 404.151,Z 348.768,A -85,B 0,C 180,E1 -11013.812,E2 -11013.812} C_VEL
LIN {X 0,Y 404.141,Z 348.768,A -85,B 0,C 180,E1 -11016.874,E2 -11016.874} C_VEL
LIN {X 0,Y 404.153,Z 348.769,A -85,B 0,C 180,E1 -11020.08,E2 -11020.08} C_VEL
LIN {X 0,Y 404.158,Z 348.759,A -85,B 0,C 180,E1 -11023.083,E2 -11023.083} C_VEL
LIN {X 0,Y 404.153,Z 348.752,A -85,B 0,C 180,E1 -11025.926,E2 -11025.926} C_VEL
LIN {X 0,Y 404.124,Z 348.767,A -85,B 0,C 180,E1 -11028.634,E2 -11028.634} C_VEL
LIN {X 0,Y 404.162,Z 348.761,A -85,B 0,C 180,E1 -11031.491,E2 -11031.491} C_VEL
LIN {X 0,Y 404.191,Z 348.758,A -85,B 0,C 180,E1 -11034.983,E2 -11034.983} C_VEL
LIN {X 0,Y 404.148,Z 348.77,A -85,B 0,C 180,E1 -11038.553,E2 -11038.553} C_VEL
LIN {X 0,Y 404.215,Z 348.817,A -85,B 0,C 180,E1 -11040.866,E2 -11040.866} C_VEL
LIN {X 0,Y 406.564,Z 359,A -85,B 0,C 180,E1 -11043.291,E2 -11043.291} C_VEL
LIN {X 0,Y 408.483,Z 369.458,A -85,B 0,C 180,E1 -11045.61,E2 -11045.61} C_VEL
LIN {X 0,Y 408.318,Z 372.363,A -85,B 0,C 180,E1 -11046.14,E2 -11046.14} C_VEL
LIN {X 0,Y 413.672,Z 398.926,A -85,B 0,C 180,E1 -11046.983,E2 -11046.983} C_VEL
LIN {X 0,Y 413.93,Z 403.704,A -85,B 0,C 180,E1 -11047.086,E2 -11047.086} C_VEL
LIN {X 0,Y 412.219,Z 509.267,A -85,B 0,C 180,E1 -11048.954,E2 -11048.954} C_VEL
LIN {X 0,Y 411.564,Z 523.94,A -85,B 0,C 180,E1 -11049.408,E2 -11049.408} C_VEL
LIN {X 0,Y 410.102,Z 531.433,A -85,B 0,C 180,E1 -11049.672,E2 -11049.672} C_VEL
LIN {X 0,Y 404.689,Z 545.818,A -85,B 0,C 180,E1 -11050.234,E2 -11050.234} C_VEL
LIN {X 0,Y 403.3,Z 551.139,A -85,B 0,C 180,E1 -11050.542,E2 -11050.542} C_VEL
LIN {X 0,Y 403.06,Z 552.889,A -85,B 0,C 180,E1 -11050.664,E2 -11050.664} C_VEL
LIN {X 0,Y 401.985,Z 564.979,A -85,B 0,C 180,E1 -11051.656,E2 -11051.656} C_VEL
LIN {X 0,Y 400.714,Z 577.337,A -85,B 0,C 180,E1 -11052.915,E2 -11052.915} C_VEL
LIN {X 0,Y 399.673,Z 587.488,A -85,B 0,C 180,E1 -11054.182,E2 -11054.182} C_VEL
LIN {X 0,Y 398.591,Z 597.567,A -85,B 0,C 180,E1 -11055.708,E2 -11055.708} C_VEL
LIN {X 0,Y 397.851,Z 605.937,A -85,B 0,C 180,E1 -11057.242,E2 -11057.242} C_VEL
LIN {X 0,Y 396.953,Z 613.932,A -85,B 0,C 180,E1 -11059.027,E2 -11059.027} C_VEL
